	// Inputs Outputs
	Digital_Inputs_NrOfObjects			: ST_CAN_Object := (Name:='Digital Inputs_NrOfObjects',				Index:=16#21C0,					Length:=1, 	Default_Value:=14);
	Digital_Inputs_Digital_Input_1		: ST_CAN_Object := (Name:='Digital Inputs_Digital Input 1',			Index:=16#21C0,	Subindex:=1,	Length:=2);
	Digital_Inputs_Digital_Input_2		: ST_CAN_Object := (Name:='Digital Inputs_Digital Input 2',			Index:=16#21C0,	Subindex:=2,	Length:=2);
	Digital_Inputs_Digital_Input_3		: ST_CAN_Object := (Name:='Digital Inputs_Digital Input 3',			Index:=16#21C0,	Subindex:=3,	Length:=2);
	Digital_Inputs_Digital_Input_4		: ST_CAN_Object := (Name:='Digital Inputs_Digital Input 4',			Index:=16#21C0,	Subindex:=4,	Length:=2);
	Digital_Inputs_Digital_Input_5		: ST_CAN_Object := (Name:='Digital Inputs_Digital Input 5',			Index:=16#21C0,	Subindex:=5,	Length:=2);
	Digital_Inputs_Digital_Input_6		: ST_CAN_Object := (Name:='Digital Inputs_Digital Input 6',			Index:=16#21C0,	Subindex:=6,	Length:=2);
	Digital_Inputs_Digital_Input_7		: ST_CAN_Object := (Name:='Digital Inputs_Digital Input 7',			Index:=16#21C0,	Subindex:=7,	Length:=2);
	Digital_Inputs_Digital_Input_8		: ST_CAN_Object := (Name:='Digital Inputs_Digital Input 8',			Index:=16#21C0,	Subindex:=8,	Length:=2);
	Digital_Inputs_Watchdog_Input		: ST_CAN_Object := (Name:='Digital Inputs_Watchdog Input',			Index:=16#21C0,	Subindex:=9,	Length:=2);
	Digital_Inputs_Watchdog_Control		: ST_CAN_Object := (Name:='Digital Inputs_Watchdog Control',		Index:=16#21C0,	Subindex:=10,	Length:=2);
	Digital_Inputs_Watchdog_Fault		: ST_CAN_Object := (Name:='Digital Inputs_Watchdog Fault',			Index:=16#21C0,	Subindex:=11,	Length:=2);
	Digital_Inputs_PWM_enabled			: ST_CAN_Object := (Name:='Digital Inputs_PWM enabled',				Index:=16#21C0,	Subindex:=12,	Length:=2);
	Digital_Inputs_STO_L				: ST_CAN_Object := (Name:='Digital Inputs_STO_L',					Index:=16#21C0,	Subindex:=13,	Length:=2);
	Digital_Inputs_HW_ID				: ST_CAN_Object := (Name:='Digital Inputs_HW ID',					Index:=16#21C0,	Subindex:=14,	Length:=2);
	Digital_Outputs_NrOfObjects			: ST_CAN_Object := (Name:='Digital Outputs_NrOfObjects',			Index:=16#21C1,					Length:=1,						Default_Value:=3);
	Digital_Outputs_Digital_Output_1	: ST_CAN_Object := (Name:='Digital Outputs_Digital Output 1',		Index:=16#21C1,	Subindex:=1,	Length:=2);
	Digital_Outputs_Digital_Output_2	: ST_CAN_Object := (Name:='Digital Outputs_Digital Output 2',		Index:=16#21C1,	Subindex:=2,	Length:=2);
	Digital_Outputs_Digital_Output_3	: ST_CAN_Object := (Name:='Digital Outputs_Digital Output 3',		Index:=16#21C1,	Subindex:=3,	Length:=2);
	Analog_Inputs_NrOfObjects			: ST_CAN_Object := (Name:='Analog Inputs_NrOfObjects',				Index:=16#21C2,					Length:=1,						Default_Value:=2);
	Analog_Inputs_Analog_In_1			: ST_CAN_Object := (Name:='Analog Inputs_Analog In 1',				Index:=16#21C2,	Subindex:=1,	Length:=2);
	Analog_Inputs_Analog_In_2			: ST_CAN_Object := (Name:='Analog Inputs_Analog In 2',				Index:=16#21C2,	Subindex:=2,	Length:=2);
	
	// Temperature
	Drive_temperature					: ST_CAN_Object := (Name:='Drive temperature', 						Index:=16#2200,					Length:=2);
	Motor_temperature					: ST_CAN_Object := (Name:='Motor temperature', 						Index:=16#2202,					Length:=2);
	
	// HEM Reset
	BiSS_Encoder_Reset					: ST_CAN_Object := (Name:='BiSS Encoder Reset', 					Index:=16#3502,					Length:=1);
	
	// Time
	Time_since_power_on					: ST_CAN_Object := (Name:='Time since power on', 					Index:=16#4008);
	
	// CAN parameters
	CAN_open_Settings_NrOfObjects		: ST_CAN_Object := (Name:='CAN open Settings_NrOfObjects', 			Index:=16#400A,					Length:=1, 						Default_Value:=2);
	CAN_open_Settings_Node_Id			: ST_CAN_Object := (Name:='CAN open Settings_Node Id', 				Index:=16#400A,	Subindex:=1,	Length:=1,	RPDO_Mappable:=TRUE,Default_Value:=2);
	CAN_open_Settings_Baud_rate			: ST_CAN_Object := (Name:='CAN open Settings_Baud rate', 			Index:=16#400A,	Subindex:=2,	Length:=1,	RPDO_Mappable:=TRUE,Default_Value:=0);
	
	// Reset
	Reset								: ST_CAN_Object := (Name:='Reset', 									Index:=16#400B,					Length:=2);
	
	// Error, warning, message
	Error_Warning_status_NrOfObjects					: ST_CAN_Object := (Name:='Error Warning status_NrOfObjects', 						Index:=16#4080,					Length:=1, Default_Value:=2);
	Error_Warning_status_Error_count					: ST_CAN_Object := (Name:='Error Warning status_Error count', 						Index:=16#4080,	Subindex:=1);
	Error_Warning_status_Warning_count					: ST_CAN_Object := (Name:='Error Warning status_Warning count', 					Index:=16#4080,	Subindex:=2);
	Message_History_NrOfObjects							: ST_CAN_Object := (Name:='Message History_NrOfObjects', 							Index:=16#4081,					Length:=1, Default_Value:=6);
	Message_History_Rx_Last_address						: ST_CAN_Object := (Name:='Message History_Rx Last address', 						Index:=16#4081,	Subindex:=1);
	Message_History_Rx_Last_message_data				: ST_CAN_Object := (Name:='Message History_Rx Last message data', 					Index:=16#4081,	Subindex:=2);
	Message_History_Rx_2nd_Last_address					: ST_CAN_Object := (Name:='Message History_Rx 2nd Last address', 					Index:=16#4081,	Subindex:=3);
	Message_History_Rx_2nd_Last_message_data			: ST_CAN_Object := (Name:='Message History_Rx 2nd Last message data',				Index:=16#4081,	Subindex:=4);
	Message_History_Rx_3rd_Last_address					: ST_CAN_Object := (Name:='Message History_Rx 3rd Last address', 					Index:=16#4081,	Subindex:=5);
	Message_History_Rx_3rd_Last_message_data			: ST_CAN_Object := (Name:='Message History_Rx 3rd Last message data',				Index:=16#4081,	Subindex:=6);
	Error_history_device_time_NrOfObjects				: ST_CAN_Object := (Name:='Error history device time_NrOfObjects',					Index:=16#4082,					Length:=1, Default_Value:=4);
	Error_history_device_time_Field_1					: ST_CAN_Object := (Name:='Error history device time_Field 1', 						Index:=16#4082,	Subindex:=1);
	Error_history_device_time_Field_2					: ST_CAN_Object := (Name:='Error history device time_Field 2', 						Index:=16#4082,	Subindex:=2);
	Error_history_device_time_Field_3					: ST_CAN_Object := (Name:='Error history device time_Field 3', 						Index:=16#4082,	Subindex:=3);
	Error_history_device_time_Field_4					: ST_CAN_Object := (Name:='Error history device time_Field 4', 						Index:=16#4082,	Subindex:=4);
	Manufacturer_Error_Message_and_Code_NrOfObjects		: ST_CAN_Object := (Name:='Manufacturer Error Message and Code_NrOfObjects', 		Index:=16#4083,					Length:=1, Default_Value:=8);
	Manufacturer_Error_Message_and_Code_Field_1_Message	: ST_CAN_Object := (Name:='Manufacturer Error Message and Code_Field 1 Message', 	Index:=16#4083,	Subindex:=1);
	Manufacturer_Error_Message_and_Code_Field_1_Code	: ST_CAN_Object := (Name:='Manufacturer Error Message and Code_Field 1 Code', 		Index:=16#4083,	Subindex:=2,	Length:=2);
	Manufacturer_Error_Message_and_Code_Field_2_Message	: ST_CAN_Object := (Name:='Manufacturer Error Message and Code_Field 2 Message', 	Index:=16#4083,	Subindex:=3);
	Manufacturer_Error_Message_and_Code_Field_2_Code	: ST_CAN_Object := (Name:='Manufacturer Error Message and Code_Field 2 Code', 		Index:=16#4083,	Subindex:=4,	Length:=2);
	Manufacturer_Error_Message_and_Code_Field_3_Message	: ST_CAN_Object := (Name:='Manufacturer Error Message and Code_Field 3 Message', 	Index:=16#4083,	Subindex:=5);
	Manufacturer_Error_Message_and_Code_Field_3_Code	: ST_CAN_Object := (Name:='Manufacturer Error Message and Code_Field 3 Code', 		Index:=16#4083,	Subindex:=6,	Length:=2);
	Manufacturer_Error_Message_and_Code_Field_4_Message	: ST_CAN_Object := (Name:='Manufacturer Error Message and Code_Field 4 Message', 	Index:=16#4083,	Subindex:=7);
	Manufacturer_Error_Message_and_Code_Field_4_Code	: ST_CAN_Object := (Name:='Manufacturer Error Message and Code_Field 4 Code', 		Index:=16#4083,	Subindex:=8,	Length:=2);
	Warning_Code_NrOfObjects							: ST_CAN_Object := (Name:='Warning Code_NrOfObjects', 								Index:=16#408A, 				Length:=1, Default_Value:=4);
	Warning_Code_Field_1								: ST_CAN_Object := (Name:='Warning Code_Field 1', 									Index:=16#408A,	Subindex:=1, 	Length:=2);
	Warning_Code_Field_2								: ST_CAN_Object := (Name:='Warning Code_Field 2', 									Index:=16#408A,	Subindex:=2, 	Length:=2);
	Warning_Code_Field_3								: ST_CAN_Object := (Name:='Warning Code_Field 3', 									Index:=16#408A,	Subindex:=3, 	Length:=2);
	Warning_Code_Field_4								: ST_CAN_Object := (Name:='Warning Code_Field 4', 									Index:=16#408A,	Subindex:=4, 	Length:=2);
	Warning_history_device_time_NrOfObjects				: ST_CAN_Object := (Name:='Warning history device time_NrOfObjects', 				Index:=16#408B, 				Length:=1, Default_Value:=4);
	Warning_history_device_time_Field_1					: ST_CAN_Object := (Name:='Warning history device time_Field 1', 					Index:=16#408B,	Subindex:=1);
	Warning_history_device_time_Field_2					: ST_CAN_Object := (Name:='Warning history device time_Field 2', 					Index:=16#408B,	Subindex:=2);
	Warning_history_device_time_Field_3					: ST_CAN_Object := (Name:='Warning history device time_Field 3', 					Index:=16#408B,	Subindex:=3);
	Warning_history_device_time_Field_4					: ST_CAN_Object := (Name:='Warning history device time_Field 4', 					Index:=16#408B,	Subindex:=4);
	Errors_Warnings_Version								: ST_CAN_Object := (Name:='Errors/Warnings Version', 								Index:=16#40BF, 				Length:=2);
END_VAR

// ---- GVLs/PDO.TcGVL
{attribute 'qualified_only'}
VAR_GLOBAL
	// Values for RPDOs
	Controlword 				AT%Q*: WORD 				:= 0;
	Mode_of_operation 			AT%Q*: E_Mode_of_Operation 	:= E_Mode_of_Operation.No_mode_active;
	Target_velocity		 		AT%Q*: DINT 				:= 0;
	Profile_velocity			AT%Q*: DINT					:= 0;
	Target_position		 		AT%Q*: DINT					:= 0;
	Target_torque		 		AT%Q*: INT					:= 0;
	vl_target_velocity	 		AT%Q*: INT					:= 0;
	
		
	// Values from TPDOs
	Statusword 					AT%I*: WORD					:= 0;
	Mode_of_operation_display	AT%I*: E_Mode_of_Operation 	:= E_Mode_of_Operation.No_mode_active;
	DC_link_circuit_voltage		AT%I*: DWORD				:= 0;
	Current_actual_value		AT%I*: INT					:= 0;
	Velocity_actual_value 		AT%I*: DINT					:= 0;
	Position_actual_value 		AT%I*: DINT					:= 0;
	Torque_actual_value 		AT%I*: INT					:= 0;
	Drive_temperature			AT%I*: INT					:= 0;
	Motor_temperature			AT%I*: INT					:= 0;
	vl_Velocity_actual_value 		AT%I*: INT					:= 0;	
END_VAR

// ---- POUs/MAIN.TcPOU
PROGRAM MAIN
VAR		
	State			: INT			:= 255;
	
	Controlmode		: E_Controlmode;
	
	Current_State	: E_Statemachine_State;
	Target_State	: E_Statemachine_State;
		
	bTaster1 AT%I*	: BOOL;
	bTaster2 AT%I*	: BOOL;
	bTaster3 AT%I*	: BOOL;
	bTaster4 AT%I*	: BOOL;
	bTaster5 AT%I*	: BOOL;
	bTaster6 AT%I*	: BOOL;
	bTaster7 AT%I*	: BOOL;
	bTaster8 AT%I*	: BOOL;
	bTaster1_Flanke	: R_TRIG;
	bTaster2_Flanke	: R_TRIG;
	bTaster3_Flanke	: R_TRIG;
	bTaster4_Flanke	: R_TRIG;
	bTaster5_Flanke	: R_TRIG;
	bTaster6_Flanke	: R_TRIG;
	bTaster7_Flanke	: R_TRIG;
	bTaster8_Flanke	: R_TRIG;
	
	
	bLED1 	AT%Q* 	: BOOL;
	bLED2 	AT%Q* 	: BOOL;
	bLED3 	AT%Q* 	: BOOL;
	bLED4 	AT%Q* 	: BOOL;
	bLED5 	AT%Q* 	: BOOL;
	bLED6 	AT%Q* 	: BOOL;
	bLED7 	AT%Q* 	: BOOL;
	bLED8 	AT%Q* 	: BOOL;
	
	CAN_Object_Testing		: FB_DS402_Object_Testing;
			
	Profile_Position_Mode	: Profile_Position_Mode;
	
	READ_Manufacturer_label	: READ_Manufacturer_label;
	
	Encoder_Alignment		: Encoder_Alignment;
	
	Homing_parameters		: ST_Homing_parameters;
	Homing_mode				: Homing_Mode;
	
	NodeID			: BYTE := 2;
	
	Data		: ARRAY [0..255] OF BYTE;
	
	SDO_READ		: FB_SDO_READ;
	ReadStart		: BOOL;
	ReadError		: DWORD;
	ReadData		: ARRAY [0..255] OF BYTE;
	
	SDO_WRITE		: FB_SDO_WRITE;
	WriteData		: ARRAY [0..255] OF BYTE;
	WriteStart		: BOOL;
	WriteError		: DWORD;

	Start_Testing	: FB_Sequenz_Testing;
	
	Position_set	: BOOL;
	
	Position_1		: DINT 	:= 0;
	Position_2		: DINT	:= 16#10000;

	Start_Merker	: BOOL;
	Finished		: BOOL;
	i				: DINT;
	
	STOP			: BOOL;
	
	Quick_Stop		: BOOL := FALSE;
	
	New_Controlword	: WORD;
		
	Fehler: DWORD;
	
	Startsequence 	: ARRAY [0..12] OF E_Test_step 	:= [E_Test_step.Switch_on_disabled,															
														E_Test_step.Velocity_window_30rpm,
														E_Test_step.Velocity_window_100ms,	
														E_Test_step.Mode_PVM,
														E_Test_step.Acceleration_1000,
														E_Test_step.Deceleration_1000,
														E_Test_step.PVM_Velocity_1000,
														E_Test_step.Ready_to_switch_on,
														E_Test_step.Switched_on,
														E_Test_step.Operation_enabled,
														E_Test_step.Wait_1000ms, 
														E_Test_step.Check_Statusword_Target_reached_200ms, 
														E_Test_step.Switch_on_disabled];
	
	Stop_Testing_SM : J_Stop_Testing_SM;
	Temp_Control_Word : WORD;
END_VAR

// Determine state
Current_State := GET_STATE(PDO.Statusword);
(*
// Show State with LEDs on IO module
bLED1 := (Current_State = E_Statemachine_State.Not_ready_to_switch_on);
bLED2 := (Current_State = E_Statemachine_State.Switch_on_disabled);
bLED3 := (Current_State = E_Statemachine_State.Ready_to_switch_on);
bLED4 := (Current_State = E_Statemachine_State.Switched_on);
bLED5 := (Current_State = E_Statemachine_State.Operation_enabled);
bLED6 := (Current_State = E_Statemachine_State.Quick_stop_active);
bLED7 := (Current_State = E_Statemachine_State.Fault_reaction_active);
bLED8 := (Current_State = E_Statemachine_State.Fault);

// Stop condition is all taster off
STOP := NOT bTaster1 AND NOT bTaster2 AND NOT bTaster3 AND NOT bTaster4 AND NOT bTaster5 AND NOT bTaster6 AND NOT bTaster7 AND NOT bTaster8;

// Reset if all taster are high
IF bTaster1 AND bTaster2 AND bTaster3 AND bTaster4 AND bTaster5 AND bTaster6 AND bTaster7 AND bTaster8 THEN
	State := 0;
END_IF

// Detect rising egdes
bTaster1_Flanke(CLK := bTaster1);
bTaster2_Flanke(CLK := bTaster2);
bTaster3_Flanke(CLK := bTaster3);
bTaster4_Flanke(CLK := bTaster4);
bTaster5_Flanke(CLK := bTaster5);	
bTaster6_Flanke(CLK := bTaster6);
bTaster7_Flanke(CLK := bTaster7);
bTaster8_Flanke(CLK := bTaster8);

*)
New_Controlword := PDO.Controlword;
Temp_Control_Word := New_Controlword;

//Stop Testing Added by Jan

	IF NOT Stop_Testing_SM.Finished THEN
		Stop_Testing_SM( JST_NodeID := NodeID,
					     JST_Start_Testing := TRUE,
						 JST_Current_State := Current_State,
						 JST_Controlword => New_Controlword);
						   
	END_IF



// Logger
GLB.Logger();
(*	


CASE State OF	
	// ********** Initial steps **********	
	0: // Idle
		CASE Controlmode OF
			E_controlmode.IO_Testmode:
				// In this mode the function are startet by digital inputs.		
				Target_State 			:= E_statemachine_state.Switch_on_disabled;
				PDO.Mode_of_operation 	:= E_Mode_of_operation.No_mode_active;
			
				IF NOT Stop THEN
					IF 		bTaster1_Flanke.Q 	THEN	
						// ************** Object test **************	
						State := 10;							
					
					ELSIF 	bTaster2_Flanke.Q 	THEN	
						// ********* Test the Start Testing ********
						State := 40;


					//ELSIF 	bTaster2_Flanke.Q 	THEN							
						// ********** Velocity Mode **********	
						//PDO.Mode_of_operation 	:= E_Mode_of_operation.Velocity_mode;
						//Target_State 			:= E_statemachine_state.Operation_enabled;
						//PDO.vl_target_velocity 	:= 1000;
						//State := 1;
						
					ELSIF 	bTaster3_Flanke.Q 	THEN
						// ********** Profile Velocity Mode **********			
						PDO.Mode_of_operation 	:= E_Mode_of_operation.Profile_velocity_mode;
						Target_State 			:= E_statemachine_state.Operation_enabled;
						PDO.Target_velocity 	:= 100000;			
						State := 1;
			
					ELSIF 	bTaster4_Flanke.Q 	THEN
						// ********** Profile Position Mode **********	
						PDO.Mode_of_operation 	:= E_Mode_of_operation.Profile_position_mode;
						Target_State 			:= E_statemachine_state.Operation_enabled;
						PDO.Profile_velocity 	:= 1000000;						
						PDO.Target_position 	:= Position_1;	
						Start_Merker 			:= TRUE;
						State := 1;
						
					ELSIF 	bTaster5_Flanke.Q 	THEN
						// ********** Profile Position Mode **********	
						PDO.Mode_of_operation 	:= E_Mode_of_operation.Profile_position_mode;
						Target_State 			:= E_statemachine_state.Operation_enabled;
						PDO.Profile_velocity 	:= 100000;
						PDO.Target_position 	:= Position_2;	
						Start_Merker 			:= TRUE;
						State := 1;
						
					//ELSIF 	bTaster6_Flanke.Q 	THEN  
						// ************* Homing mode **************		
					//	Homing_parameters.Homing_mode := E_Homing_mode.Homing_on_current_position;			
					//	State := 20;				
						
					ELSIF 	bTaster6_Flanke.Q 	THEN	
						// Open / Close Logger File				
						IF GLB.Logger.IsOpen THEN 
							GLB.Logger(CloseFlag := TRUE);
						ELSE
							GLB.Logger(OpenFlag := TRUE);				
						END_IF								
					
					ELSIF 	bTaster7_Flanke.Q	THEN
						// Test: Write Logger Message						
						GLB.Logger(Message:= 'Hallo');	

					ELSIF 	bTaster8_Flanke.Q	THEN
						// Test: Save Logger Message						
						GLB.Logger(SaveFlag := TRUE);
						
					END_IF			
				END_IF					
				New_Controlword := CONTROLWORD_STATE_CHANGE(Current_State, Target_State);	
						
				
			E_Controlmode.Manual:
				// The user have to set the pdo values or the target state manually.
				State := 255;
			
		END_CASE
		
		
	1: // Start process
		IF 	STOP THEN	
			Target_State := E_statemachine_state.Switch_on_disabled;
			State := 3;	
		ELSIF Current_State = E_statemachine_state.Operation_enabled THEN 	
			State := 2;			
		END_IF;		
	
		New_Controlword := CONTROLWORD_STATE_CHANGE(Current_State, Target_State);	
				
		
	2: // Mode specific
		New_Controlword := CONTROLWORD_STATE_CHANGE(Current_State, Target_State);
	
		CASE PDO.Mode_of_operation OF				
			E_Mode_of_operation.Profile_position_mode:
				Profile_Position_Mode(Current_State:=Current_State, Statusword:=PDO.Statusword, Controlword:=New_Controlword, Start:=Start_Merker, Finished=>Finished);
				
				
		END_CASE
				
		IF STOP THEN 
			Target_State := E_statemachine_state.Switch_on_disabled;
			New_Controlword := CONTROLWORD_STATE_CHANGE(Current_State, Target_State);	
			State := 3; 
		END_IF
					
		
	3:	// Stop process
		Target_State := E_statemachine_state.Switch_on_disabled;	
		New_Controlword := CONTROLWORD_STATE_CHANGE(Current_State, Target_State);			
		IF Current_State = E_statemachine_state.Switch_on_disabled THEN	State := 0;	END_IF
		
		
	10:	// ********** CAN Object Testing **********	
		CAN_Object_Testing(Start := TRUE);	
		State := State + 1;

	11: // Wait for finish
		CAN_Object_Testing(Start := FALSE);		
		IF CAN_Object_Testing.Finished AND STOP THEN	
			State := 0;	
		END_IF
			
		
	20:	// ************* Homing mode **************
		Homing_mode(NodeID:=NodeID, Start:=TRUE, Current_State:=Current_State, Statusword:=PDO.Statusword, Homing_parameters:=Homing_parameters, Controlword=>New_Controlword, Mode_of_operation=>PDO.Mode_of_operation);
		State := State + 1;
	
	21: // Wait for finish
		Homing_mode(Start:=FALSE, Current_State:=Current_State, Statusword:=PDO.Statusword, Controlword=>New_Controlword);	
		IF Homing_mode.Finished THEN
			State := 0;
		END_IF
		
		
	30:	// ********** Encoder Alignment ***********	
		Encoder_Alignment(Start:=TRUE, Current_State:=Current_State, Statusword:=PDO.Statusword, Controlword=>New_Controlword);
		State := State + 1;
	
	31: // Wait for finish
		Encoder_Alignment(Start:=FALSE, Current_State:=Current_State, Statusword:=PDO.Statusword, Controlword=>New_Controlword);	
		IF Encoder_Alignment.Finished THEN
			State := 0;
		END_IF

		
	40:	// Test the Start Testing		
		Start_Testing(Start:=TRUE, Sequence_Name:='Test Sequence', Step_list:=Startsequence);
		State := State + 1;
	
	41: // Wait for finish
		Start_Testing(Start:=FALSE);
		New_Controlword := PDO.Controlword;		
		IF Start_Testing.Finished THEN
			State := 0;
		END_IF

		
	255: // **************** Init *****************
		GLB.Logger(OpenFlag:=TRUE);
		State := 0;
	
		
	ELSE	// Reset to Idle
		State := 0;
	
END_CASE	
*)

// Write the new Controlword
PDO.Controlword := New_Controlword;

END_PROGRAM

// ---- POUs/CAN_Object_Testing.TcPOU
FUNCTION_BLOCK CAN_Object_Testing
VAR_INPUT
	NodeID			: BYTE; (* This Port No. addresses the CANopen Node (see System Manager) *)
	Start			: BOOL;
END_VAR
VAR_OUTPUT
	Finished		: BOOL;
END_VAR
VAR_IN_OUT
	CAN_Objects		: ARRAY [*] OF ST_CAN_Object;
END_VAR
VAR
	State			: BYTE := 0;
	Index			: DINT := 0;
	i				: BYTE := 0;
	
	Data		: ARRAY [0..255] OF BYTE;
	
	NMT_WRITE		: FB_NMT_WRITE;
	SDO_READ		: FB_SDO_READ;
	SDO_WRITE		: FB_SDO_WRITE;	
			
	RPDO_Nr				: BYTE := 3;	
	RPDO_Current_Number	: BYTE := 0;
	RPDO_Current_Mapped	: DWORD := 0;	
	
	TPDO_Nr				: BYTE := 3;
	TPDO_Current_Number	: BYTE := 0;
	TPDO_Current_Mapped	: DWORD := 0;
END_VAR

IF Start AND State = 255 THEN 
	State := 0;
END_IF

SDO_READ(StartReading:=FALSE);
SDO_WRITE(StartWriting:=FALSE);
NMT_WRITE(StartWriting:=FALSE);


CASE State OF	
	// ********** Initial steps **********	
	0: // NMT Set to Preoperational
		IF Start THEN
			NMT_WRITE(
				AdsNetID	:= GLB.ADSNetID_CAN,
				PortNr		:= 16#1000 + GLB.NodeID,
				ADSSTATE	:= ADSSTATE_RUN, 
				DEVSTATE	:= 0,
				StartWriting:=TRUE			
			);	
			State := State + 1;			
		END_IF
		
	1: // Wait for finish			
			IF NMT_WRITE.WriteDataFinished THEN
				Index := 0;	
				State := State + 1;	
			END_IF

			
	2:	// RPDO disable
		Data[3] := 16#80;
		Data[2] := 0;			
		Data[1] := RPDO_Nr + 1;
		Data[0] := NodeID;	
			
		SDO_WRITE(
			ADSNetID		:= GLB.ADSNetID_CAN,
			PortNr 		 	:= 16#1000 + GLB.NodeID,
			CO_Index 	 	:= 16#1400 + RPDO_Nr,
			CO_SubIndex  	:= 1,
			DataLength 	 	:= 4,
			StartWriting 	:= TRUE,
			WriteData 	 	:= Data );
		State := State + 1;	
		
	3: // Wait for finish
		IF SDO_WRITE.WriteDataFinished THEN
			State := State + 1;
		END_IF	
		
		
	4:	// RPDO Current Number of mapped objects
		SDO_READ(
			ADSNetID		:= GLB.ADSNetID_CAN,				
			PortNr 		 	:= 16#1000 + GLB.NodeID,
			CO_Index 		:= 16#1600 + RPDO_Nr,
			CO_SubIndex 	:= 0,
			DataLength 		:= 1,
			StartReading	:= TRUE	);
		State := State + 1;	
		
	5: // Wait for finish
		IF SDO_READ.ReadDataAvailable THEN
			RPDO_Current_Number := SDO_READ.ReadData[0];
			State := State + 1;
		END_IF
		
	
	6:	// RPDO Current mapped object
		SDO_READ(
			ADSNetID		:= GLB.ADSNetID_CAN,				
			PortNr 		 	:= 16#1000 + GLB.NodeID,
			CO_Index 		:= 16#1600 + RPDO_Nr,
			CO_SubIndex 	:= 1,
			DataLength 		:= 4,
			StartReading	:= TRUE);
		State := State + 1;	
		
	7: // Wait for finish
		IF SDO_READ.ReadDataAvailable THEN
			RPDO_Current_Mapped := SHL(BYTE_TO_DWORD(SDO_READ.ReadData[3]),24) + SHL(BYTE_TO_DWORD(SDO_READ.ReadData[2]),16) + SHL(BYTE_TO_DWORD(SDO_READ.ReadData[1]),8) + BYTE_TO_DWORD(SDO_READ.ReadData[0]);								
			State := State + 1;
		END_IF		
			
		
	8:	// TPDO disable
		Data[3] := 16#80;
		Data[2] := 0;			
		Data[1] := TPDO_Nr;
		Data[0] := NodeID + 16#80;	
			
		SDO_WRITE(
			ADSNetID		:= GLB.ADSNetID_CAN,
			PortNr 		 	:= 16#1000 + GLB.NodeID,
			CO_Index 	 	:= 16#1800 + TPDO_Nr,
			CO_SubIndex  	:= 1,
			DataLength 	 	:= 4,
			StartWriting 	:= TRUE,
			WriteData 	 	:= Data );		
		State := State + 1;	
		
	9: // Wait for finish
		IF SDO_WRITE.WriteDataFinished THEN
			State := State + 1;
		END_IF	
		

	10:	// TPDO Current Number of mapped objects
		SDO_READ(
			ADSNetID		:= GLB.ADSNetID_CAN,				
			PortNr 		 	:= 16#1000 + GLB.NodeID,
			CO_Index 		:= 16#1A00 + TPDO_Nr,
			CO_SubIndex 	:= 0,
			DataLength 		:= 1,
			StartReading	:= TRUE	);		
		State := State + 1;	
		
	11: // Wait for finish
		IF SDO_READ.ReadDataAvailable THEN
			TPDO_Current_Number := SDO_READ.ReadData[0];			
			State := State + 1;
		END_IF
		

	12:	// TPDO Current mapped object
		SDO_READ(
			ADSNetID		:= GLB.ADSNetID_CAN,				
			PortNr 		 	:= 16#1000 + GLB.NodeID,
			CO_Index 		:= 16#1A00 + TPDO_Nr,
			CO_SubIndex 	:= 1,
			DataLength 		:= 4,
			StartReading	:= TRUE	);		
		State := State + 1;	
		
	13: // Wait for finish
		IF SDO_READ.ReadDataAvailable THEN
			TPDO_Current_Mapped := SHL(BYTE_TO_DWORD(SDO_READ.ReadData[3]),24) + SHL(BYTE_TO_DWORD(SDO_READ.ReadData[2]),16) + SHL(BYTE_TO_DWORD(SDO_READ.ReadData[1]),8) + BYTE_TO_DWORD(SDO_READ.ReadData[0]);							
			State := 16;
		END_IF		
		
		
		
	// ********** Test steps **********
	16:	// Init
		IF CAN_Objects[Index].Length_Tested THEN 
			CAN_Objects[Index].Length_Tested := FALSE;
			CAN_Objects[Index].Length_Error := 0;
		ELSE
			CAN_Objects[Index].Length_Target := CAN_Objects[Index].Length; 
		END_IF
		
		IF CAN_Objects[Index].Readable_Tested THEN 
			CAN_Objects[Index].Readable_Tested := FALSE;
			CAN_Objects[Index].Readable_Error := 0;
			CAN_Objects[Index].Read_Value := 0;
		ELSE
			CAN_Objects[Index].Readable_Target := CAN_Objects[Index].Readable;
		END_IF
		
		IF CAN_Objects[Index].Writable_Tested THEN 
	    	CAN_Objects[Index].Writable_Tested := FALSE;
			CAN_Objects[Index].Writable_Error := 0; 
			CAN_Objects[Index].Write_Value := 0;
		ELSE		
			CAN_Objects[Index].Writable_Target := CAN_Objects[Index].Writable;
		END_IF
				
		IF CAN_Objects[Index].RPDO_Mappable_Tested THEN 
	    	CAN_Objects[Index].RPDO_Mappable_Tested := FALSE;
			CAN_Objects[Index].RPDO_Mappable_Error := 0; 
		ELSE		
			CAN_Objects[Index].RPDO_Mappable_Target := CAN_Objects[Index].RPDO_Mappable;
		END_IF
		
		IF CAN_Objects[Index].TPDO_Mappable_Tested THEN 
	    	CAN_Objects[Index].TPDO_Mappable_Tested := FALSE;
			CAN_Objects[Index].TPDO_Mappable_Error := 0; 
		ELSE		
			CAN_Objects[Index].TPDO_Mappable_Target := CAN_Objects[Index].TPDO_Mappable;
		END_IF	

		State := State + 1;
			
		
	17:	// Read Test
		SDO_READ(
			ADSNetID		:= GLB.ADSNetID_CAN,				
			PortNr 		 	:= 16#1000 + GLB.NodeID,
			CO_Index 		:= CAN_Objects[Index].Index,
			CO_SubIndex 	:= CAN_Objects[Index].Subindex,
			DataLength 		:= CAN_Objects[Index].Length,
			StartReading	:= TRUE	);		
		State := State + 1;
		
	18: // Read Test, wait for finish
		IF SDO_READ.ReadDataAvailable THEN
			CAN_Objects[Index].Readable_Tested := TRUE;
			CAN_Objects[Index].Read_Value := SHL(BYTE_TO_DWORD(SDO_READ.ReadData[3]),24) + SHL(BYTE_TO_DWORD(SDO_READ.ReadData[2]),16) + SHL(BYTE_TO_DWORD(SDO_READ.ReadData[1]),8) + BYTE_TO_DWORD(SDO_READ.ReadData[0]);	
			CAN_Objects[Index].Readable_Error := SDO_READ.Error;
			
			// LENGTH setzen !!!	
								
			State := State + 1;
		END_IF
	
		
	19:	// Write Test
		IF CAN_Objects[Index].Write_Value_Usage THEN CAN_Objects[Index].Write_Value := CAN_Objects[Index].Read_Value; END_IF
		FOR i := 0 TO CAN_Objects[Index].Length - 1 DO
			Data[i] := DWORD_TO_BYTE(SHR(CAN_Objects[Index].Write_Value, (8*i)));
		END_FOR;
			
		SDO_WRITE(
			ADSNetID	:= GLB.ADSNetID_CAN,
			PortNr 		 := 16#1000 + GLB.NodeID,
			CO_Index 	 := CAN_Objects[Index].Index,
			CO_SubIndex  := CAN_Objects[Index].Subindex,
			DataLength 	 := CAN_Objects[Index].Length,
			StartWriting := TRUE,
			WriteData 	 := Data );		
		State := State + 1;
			
	20: // Write Test, wait for finish
		IF SDO_WRITE.WriteDataFinished THEN
			CAN_Objects[Index].Writable_Tested := TRUE;
			CAN_Objects[Index].Write_Value := SHL(BYTE_TO_DWORD(SDO_Write.WriteData[3]),24) + SHL(BYTE_TO_DWORD(SDO_Write.WriteData[2]),16) + SHL(BYTE_TO_DWORD(SDO_Write.WriteData[1]),8) + BYTE_TO_DWORD(SDO_Write.WriteData[0]);				
			CAN_Objects[Index].Writable_Error := SDO_WRITE.Error;
			
			
			// Falls Read-Test nicht erfolgreich -> LENGTH hier setzen !!!	
			
		
			State := State + 1;
		END_IF

		
	21: // RPDO test	
		Data[0] := CAN_Objects[Index].Length * 8;
		Data[1] := CAN_Objects[Index].SubIndex;
		Data[2] := DWORD_TO_BYTE(CAN_Objects[Index].Index);
		Data[3] := DWORD_TO_BYTE(SHR(CAN_Objects[Index].Index,8));
			
		SDO_WRITE(
			ADSNetID	:= GLB.ADSNetID_CAN,
			PortNr 		 := 16#1000 + GLB.NodeID,
			CO_Index 	 := 16#1600 + RPDO_Nr,
			CO_SubIndex  := 1,
			DataLength 	 := 4,
			StartWriting := TRUE,
			WriteData 	 := Data );	
		State := State + 1;
			
	22: // RPDO test, wait for finish
		IF SDO_WRITE.WriteDataFinished THEN
			CAN_Objects[Index].RPDO_Mappable_Tested := TRUE;
			CAN_Objects[Index].RPDO_Mappable_Error := SDO_WRITE.Error;
									
			State := State + 1;
		END_IF	

				
	23: // TPDO test
		// Value for TPDO test is the same like RPDO test
 
		SDO_WRITE(
			ADSNetID	:= GLB.ADSNetID_CAN,
			PortNr 		 := 16#1000 + GLB.NodeID,
			CO_Index 	 := 16#1A00 + TPDO_Nr,
			CO_SubIndex  := 1,
			DataLength 	 := 4,
			StartWriting := TRUE,
			WriteData 	 := Data );	
		State := State + 1;
			
	24: // TPDO test, wait for finish
		IF SDO_WRITE.WriteDataFinished THEN
			CAN_Objects[Index].TPDO_Mappable_Tested := TRUE;
			CAN_Objects[Index].TPDO_Mappable_Error := SDO_WRITE.Error;
			
			State := State + 1;
		END_IF
		
		
	25: // Next object
		CAN_Objects[Index].Error := (CAN_Objects[Index].Readable_Error > 0) OR (CAN_Objects[Index].Writable_Error > 0) OR (CAN_Objects[Index].RPDO_Mappable_Error > 0) OR (CAN_Objects[Index].TPDO_Mappable_Error > 0);
			
		IF Index < UPPER_BOUND(CAN_Objects,1) THEN
			Index := Index + 1;
			State := 16;
		ELSE
			State := 128;
		END_IF
	
		
	// ********** Ending steps **********		
	128: // RPDO Reset mapped object
		Data[0] := DWORD_TO_BYTE(RPDO_Current_Mapped);
		Data[1] := DWORD_TO_BYTE(SHR(RPDO_Current_Mapped,8));
		Data[2] := DWORD_TO_BYTE(SHR(RPDO_Current_Mapped,16));
		Data[3] := DWORD_TO_BYTE(SHR(RPDO_Current_Mapped,24));
		SDO_WRITE(
			ADSNetID		:= GLB.ADSNetID_CAN,			
			PortNr 		 	:= 16#1000 + GLB.NodeID,
			CO_Index 		:= 16#1600 + TPDO_Nr,
			CO_SubIndex 	:= 1,
			DataLength 		:= 4,
			StartWriting	:= TRUE,
			WriteData 	 	:= Data );
		State := State + 1;
			
	129: // RPDO Reset mapped object, wait for finish		
		IF SDO_WRITE.WriteDataFinished THEN
			State := State + 1;
		END_IF		
			
		
	130: // RPDO Reset Number of mapped objects
		Data[0] := RPDO_Current_Number;
			
		SDO_WRITE(
			ADSNetID		:= GLB.ADSNetID_CAN,
			PortNr 		 	:= 16#1000 + GLB.NodeID,
			CO_Index 		:= 16#1600 + RPDO_Nr,
			CO_SubIndex 	:= 0,
			DataLength 		:= 1,
			StartWriting 	:= TRUE,
			WriteData 	 	:= Data );
		State := State + 1;
			
	131: // RPDO Reset Number of mapped objects, wait for finish			
		IF SDO_WRITE.WriteDataFinished THEN
			State := State + 1;
		END_IF			

		
	132: // RPDO reactivate
		Data[3] := 0;
		Data[2] := 0;			
		Data[1] := RPDO_Nr + 1;
		Data[0] := NodeID;	
			
		SDO_WRITE(
			ADSNetID	:= GLB.ADSNetID_CAN,
			PortNr 		 := 16#1000 + GLB.NodeID,
			CO_Index 	 := 16#1400 + RPDO_Nr,
			CO_SubIndex  := 1,
			DataLength 	 := 4,
			StartWriting := TRUE,
			WriteData 	 := Data );
		State := State + 1;
			
	133: // RPDO reactivate, wait for finish	
		IF SDO_WRITE.WriteDataFinished THEN
			State := State + 1;
		END_IF	
		
		
	134: // TPDO Reset mapped object
		Data[0] := DWORD_TO_BYTE(TPDO_Current_Mapped);
		Data[1] := DWORD_TO_BYTE(SHR(TPDO_Current_Mapped,8));
		Data[2] := DWORD_TO_BYTE(SHR(TPDO_Current_Mapped,16));
		Data[3] := DWORD_TO_BYTE(SHR(TPDO_Current_Mapped,24));
		
		SDO_WRITE(
			ADSNetID		:= GLB.ADSNetID_CAN,			
			PortNr 		 	:= 16#1000 + GLB.NodeID,
			CO_Index 		:= 16#1A00 + TPDO_Nr,
			CO_SubIndex 	:= 1,
			DataLength 		:= 4,
			StartWriting	:= TRUE,
			WriteData 	 	:= Data );
		State := State + 1;
			
	135: // TPDO Reset mapped object, wait for finish	
		IF SDO_WRITE.WriteDataFinished THEN
			State := State + 1;
		END_IF			
			
		
	136:// TPDO Reset Number of mapped objects
		Data[0] := TPDO_Current_Number;
			
		SDO_WRITE(
			ADSNetID		:= GLB.ADSNetID_CAN,
			PortNr 		 	:= 16#1000 + GLB.NodeID,
			CO_Index 		:= 16#1A00 + RPDO_Nr,
			CO_SubIndex 	:= 0,
			DataLength 		:= 1,
			StartWriting 	:= TRUE,
			WriteData 	 	:= Data );
		State := State + 1;
			
	137: // TPDO Reset Number of mapped objects, wait for finish	
		IF SDO_WRITE.WriteDataFinished THEN
			State := State + 1;
		END_IF			

		
	138: // TPDO reactivate
		Data[3] := 0;
		Data[2] := 0;			
		Data[1] := TPDO_Nr;
		Data[0] := NodeID + 16#80;	
			
		SDO_WRITE(
			ADSNetID	:= GLB.ADSNetID_CAN,
			PortNr 		 := 16#1000 + GLB.NodeID,
			CO_Index 	 := 16#1400 + RPDO_Nr,
			CO_SubIndex  := 1,
			DataLength 	 := 4,
			StartWriting := TRUE,
			WriteData 	 := Data );
		State := State + 1;
			
	139: // TPDO reactivate, wait for finish	
		IF SDO_WRITE.WriteDataFinished THEN
			State := State + 1;
		END_IF	
						
	
	140: // NMT Set to operational
		NMT_WRITE(
			ADSNetID	:= GLB.ADSNetID_CAN,
			PORTNr		:= 16#1000 + GLB.NodeID,
			ADSSTATE	:= ADSSTATE_RUN,
			DEVSTATE	:= 1,
			StartWriting:=TRUE );	
		State := State + 1;
			
	141: // RPDO Reset Number of mapped objects, wait for finish	
		IF NMT_WRITE.WriteDataFinished THEN
			State := 255;	
		END_IF

		
	// ********** End **********
	ELSE	// Tests finished	
		Finished := TRUE;
		State := 255;
			
END_CASE

END_FUNCTION_BLOCK

// ---- POUs/FB/Basic/FB_NMT_WRITE.TcPOU
FUNCTION_BLOCK FB_NMT_WRITE
VAR_INPUT
	ADSNetID		: STRING(23); 	(* The AMSNetID addresses the EL6751. Can be empty if only one local single channel card is present*)
	PortNr			: WORD; 		(* The Port No. addresses the CANopen Node (see System Manager) *)
	ADSSTATE		: UINT; 		(* This is the value of the ADS state (ADSSTATE_RUN (=5) or ADSSTATE_STOP (=6)*)
	DEVSTATE		: UINT;			(* This is the value of the wanted device state (ADSSTATE_RUN -> 1 = OP, 0 = PREOP or ADSSTATE_STOP -> 0 = STOP)*)
	StartWriting	: BOOL; 		(* only reset to FALSE after WriteDataFinished=TRUE*)
END_VAR
VAR_OUTPUT
	WriteDataFinished	: BOOL;
	Error			: DWORD;
END_VAR
VAR
	state			: BYTE := 0;
	ADSWRTCTL		: ADSWRTCTL;
	NMTData			: ARRAY[0..1] OF BYTE; (*This array contains the data to be written to the CANopen Object	Dictionary*)
END_VAR

CASE
state OF
0:
	IF StartWriting THEN
		WriteDataFinished := FALSE;
		Error := 0;
		ADSWRTCTL(
			NetID		:= ADSNetID,
			PORT		:= PortNr,
			ADSSTATE	:= ADSSTATE,
			DEVSTATE	:= DEVSTATE,
			LEN			:= 2,
			SRCADDR		:= ADR(NMTData),
			WRITE		:= TRUE,
			TMOUT 		:= T#100MS
		);	
		IF ADSWRTCTL.err THEN
			state := 2;
			WriteDataFinished := TRUE;
			Error := ADSWRTCTL.ErrId;
		ELSE
			state := 1;
		END_IF
	ELSE
		ADSWRTCTL(
			NetID		:= ADSNetID,
			PORT		:= PortNr,
			ADSSTATE	:= ADSSTATE, 
			DEVSTATE	:= DEVSTATE,
			LEN			:= 2, 
			SRCADDR		:= ADR(NMTData),
			WRITE		:= FALSE,
			TMOUT 		:= T#1S
		);
	END_IF
	
1:
	ADSWRTCTL(WRITE:= FALSE);
	IF ADSWRTCTL.err THEN
		state := 2;
		WriteDataFinished := TRUE;
		Error := ADSWRTCTL.ErrId;
	ELSE
		IF NOT ADSWRTCTL.busy THEN
			state := 2;
			WriteDataFinished := TRUE;
		END_IF
	END_IF
	
2:
	ADSWRTCTL(WRITE:= FALSE);
	state := 0;
END_CASE

END_FUNCTION_BLOCK

// ---- POUs/FB/Basic/FB_SDO_READ.TcPOU
FUNCTION_BLOCK FB_SDO_READ
VAR_INPUT
	ADSNetID		: STRING(23); 	(* The AMSNetID addresses the EL6751. Can be empty if only one local single channel card is present*)
	PortNr			: WORD;	 		(* This Port No. addresses the CANopen Node (see System Manager) *)
	CO_Index		: DWORD; 		(* This is the Index of the CANopen Object Dictionary Entry*)
	CO_SubIndex		: DWORD; 		(* This is the Sub-Index of the CANopen Object Dictionary Entry*)
	DataLength		: DWORD; 		(* This is the Length of the CANopen Object Dictionary Entry*)
	StartReading	: BOOL;  		(* only reset to FALSE after ReadDataAvailable=TRUE*)
END_VAR
VAR_OUTPUT
	ReadData		: ARRAY[0..255] OF BYTE;
	ReadDataAvailable	: BOOL;
	Error			: DWORD;
END_VAR
VAR
	state			: BYTE 	:= 0;
	ADSREAD			: ADSREAD;
END_VAR

CASE
state OF
0:
	IF StartReading THEN
		ReadDataAvailable := FALSE;
		Error := 0;
		ADSRead(
			NETID		:= ADSNetID,
			PORT		:= PortNr,
			IDXGRP		:= CO_Index,
			IDXOFFS		:= CO_SubIndex,
			LEN			:= DataLength,
			DESTADDR	:= ADR(ReadData),
			READ		:= TRUE,
			TMOUT		:= T#100MS
		);

		IF ADSRead.err THEN
			state := 2;
			ReadDataAvailable := TRUE;
			Error := ADSRead.ErrId;
		ELSE
			state := 1;
		END_IF
	ELSE
		ADSRead(
			NETID		:= ADSNetID,
			PORT		:= PortNr,
			IDXGRP		:= CO_Index,
			IDXOFFS		:= CO_SubIndex,
			LEN			:= DataLength,
			DESTADDR	:= ADR(ReadData),
			READ		:= FALSE,
			TMOUT 		:= T#100MS
		);
	END_IF
	
1:
	ADSRead(READ:= FALSE);
	IF ADSRead.err THEN
		state := 2;
		ReadDataAvailable := TRUE;
		Error := ADSRead.ErrId;
	ELSE
		IF NOT ADSRead.busy THEN
			state := 2;
			ReadDataAvailable := TRUE;
		END_IF
	END_IF
	
2:
	ADSRead(READ:= FALSE);
	state := 0;
	
END_CASE

END_FUNCTION_BLOCK

// ---- POUs/FB/Basic/FB_SDO_WRITE.TcPOU
FUNCTION_BLOCK FB_SDO_WRITE
VAR_INPUT
	ADSNetID		: STRING(23); 	(* The AMSNetID addresses the EL6751. Can be empty if only one local single channel card is present*)
	PortNr			: WORD; 		(* The Port No. addresses the CANopen Node (see System Manager) *)
	CO_Index		: DWORD; 		(* This is the Index of the CANopen Object Dictionary Entry*)
	CO_SubIndex		: DWORD; 		(* This is the Sub-Index of the CANopen Object Dictionary Entry*)
	DataLength		: DWORD; 		(* This is the Length of the CANopen Object Dictionary Entry*)
	StartWriting	: BOOL; 		(* only reset to FALSE after WriteDataFinished=TRUE*)
	WriteData		: ARRAY[0..255] OF BYTE; (*This array contains the data to be written to the CANopen Object	Dictionary*)
END_VAR
VAR_OUTPUT
	WriteDataFinished	: BOOL;
	Error			: DWORD;
END_VAR
VAR
	state			: BYTE := 0;
	ADSWRITE		: ADSWRITE;
END_VAR

CASE
state OF
0:
	IF StartWriting THEN
		WriteDataFinished := FALSE;
		Error := 0;
		ADSWrite(
			NETID	:= ADSNetID,
			PORT	:= PortNr,
			IDXGRP	:= CO_Index,
			IDXOFFS	:= CO_SubIndex,
			LEN		:= DataLength,
			SRCADDR	:= ADR(WriteData),
			WRITE	:= TRUE,
			TMOUT 	:= T#100MS
		);
		IF ADSWrite.err THEN
			state := 2;
			WriteDataFinished := TRUE;
			Error := ADSWrite.ErrId;
		ELSE
			state := 1;
		END_IF
	ELSE
		ADSWrite(
			NETID	:= '',
			PORT	:= PortNr,
			IDXGRP	:= CO_Index,
			IDXOFFS	:= CO_SubIndex,
			LEN		:= DataLength,
			SRCADDR	:= ADR(WriteData),
			WRITE	:= FALSE,
			TMOUT 	:= T#100MS
		);
	END_IF
	
1:
	ADSWrite(WRITE:= FALSE);
	IF ADSWrite.err THEN
		state := 2;
		WriteDataFinished := TRUE;
		Error := ADSWrite.ErrId;
	ELSE
		IF NOT ADSWrite.busy THEN
			state := 2;
			WriteDataFinished := TRUE;
		END_IF
	END_IF
	
2:
	ADSWrite(WRITE:= FALSE);
	state := 0;
END_CASE

END_FUNCTION_BLOCK

// ---- POUs/FB/FB_DS402_Object_Testing.TcPOU
FUNCTION_BLOCK FB_DS402_Object_Testing
VAR_INPUT
	Start			: BOOL;
END_VAR
VAR_OUTPUT
	Finished		: BOOL;
	Error			: BOOL := FALSE;
END_VAR
VAR
	State			: BYTE := 0;
	Index			: DINT := 0;
	
	NMT_WRITE		: FB_NMT_WRITE;
	
	SDO_READ		: FB_SDO_READ;
	ReadData		: ARRAY [0..255] OF BYTE;
	
	SDO_WRITE		: FB_SDO_WRITE;
	WriteData		: ARRAY [0..255] OF BYTE;		
			
	RPDO_Nr				: BYTE := 3;	
	RPDO_Current_Number	: BYTE := 0;
	RPDO_Current_Mapped	: DWORD := 0;	
	
	TPDO_Nr				: BYTE := 3;
	TPDO_Current_Number	: BYTE := 0;
	TPDO_Current_Mapped	: DWORD := 0;
	
	
	Object_List_Testing	: FB_Object_List_Testing;
	
	
	Objects_general			: ARRAY [0..11] OF ST_CAN_Object := [DS402_Object_List.Abort_connection_option_code,
																 DS402_Object_List.Error_code,
																 DS402_Object_List.Controlword,
																 DS402_Object_List.Statusword,
																 DS402_Object_List.Quick_stop_option_code,
																 DS402_Object_List.Shutdown_option_code,
																 DS402_Object_List.Disable_operation_option_code,
																 DS402_Object_List.Halt_option_code,
																 DS402_Object_List.Fault_reaction_option_code,
																 DS402_Object_List.Modes_of_operation,
																 DS402_Object_List.Modes_of_operation_display,
																 DS402_Object_List.Supported_drive_modes];
		
	Objects_Factor_group	: ARRAY [0..25] OF ST_CAN_Object := [DS402_Object_List.Position_encoder_resolution_Highest_sub_index_supported,
																 DS402_Object_List.Position_encoder_resolution_Encoder_increments,
																 DS402_Object_List.Position_encoder_resolution_Motor_revolutions,
																 DS402_Object_List.Velocity_encoder_resolution_Highest_sub_index_supported,
																 DS402_Object_List.Velocity_encoder_resolution_Encoder_increments,
																 DS402_Object_List.Velocity_encoder_resolution_Motor_revolutions,
																 DS402_Object_List.Gear_ratio_Highest_sub_index_supported,
																 DS402_Object_List.Gear_ratio_Motor_shaft_revolutions,
																 DS402_Object_List.Gear_ratio_Driving_shaft_revolutions,
																 DS402_Object_List.Feed_constant_Highest_sub_index_supported,
																 DS402_Object_List.Feed_constant_Feed,
																 DS402_Object_List.Feed_constant_Shaft_Revolution,
																 DS402_Object_List.Velocity_Factor_Highest_sub_index_supported,
																 DS402_Object_List.Velocity_Factor_Numerator,
																 DS402_Object_List.Velocity_Factor_Divisor,
																 DS402_Object_List.Acceleration_Factor_Highest_sub_index_supported,
																 DS402_Object_List.Acceleration_Factor_Numerator,
																 DS402_Object_List.Acceleration_Factor_Divisor,
																 DS402_Object_List.Jerk_factor_Factor_Highest_sub_index_supported,
																 DS402_Object_List.Jerk_factor_Factor_Numerator,
																 DS402_Object_List.Jerk_factor_Factor_Divisor,
																 DS402_Object_List.Polarity,
																 DS402_Object_List.SI_unit_postion,
																 DS402_Object_List.SI_unit_velocity,
																 DS402_Object_List.SI_unit_acceleration,
																 DS402_Object_List.SI_unit_jerk];
							
	Objects_Position_control: ARRAY [0..10] OF ST_CAN_Object := [DS402_Object_List.Position_demand_value,
															 	 DS402_Object_List.Position_actual_internal_value,
																 DS402_Object_List.Position_actual_value,
																 DS402_Object_List.Following_error_window,
																 DS402_Object_List.Following_error_time_out,
																 DS402_Object_List.Position_window,
																 DS402_Object_List.Position_window_time,
																 DS402_Object_List.Position_option_code,
																 DS402_Object_List.Following_error_actual_value,
																 DS402_Object_List.Control_effort,
																 DS402_Object_List.Position_demand_integral_value];								
	
	Objects_PPM				: ARRAY [0..20] OF ST_CAN_Object := [DS402_Object_List.Target_position,
															 	 DS402_Object_List.Position_range_limit_Highest_sub_index_supported,
																 DS402_Object_List.Position_range_limit_Min_position_range_limit,
																 DS402_Object_List.Position_range_limit_Max_position_range_limit,
																 DS402_Object_List.Software_position_limit_Highest_sub_index_supported,
																 DS402_Object_List.Software_position_limit_Min_position_limit,
																 DS402_Object_List.Software_position_limit_Max_position_limit,
																 DS402_Object_List.Polarity,
																 DS402_Object_List.Max_profile_velocity,
																 DS402_Object_List.Profile_velocity,
																 DS402_Object_List.End_velocity,
																 DS402_Object_List.Profile_acceleration,
																 DS402_Object_List.Profile_deceleration,
																 DS402_Object_List.Quick_stop_deceleration,
																 DS402_Object_List.Motion_profile_type,
																 DS402_Object_List.Profile_jerk_use,
																 DS402_Object_List.Profile_jerk_Highest_sub_index_supported,
																 DS402_Object_List.Profile_jerk_1,
																 DS402_Object_List.Max_acceleration,
																 DS402_Object_List.Max_deceleration];

	Objects_VM				: ARRAY [0..20] OF ST_CAN_Object := [DS402_Object_List.vl_target_velocity,
															 	 DS402_Object_List.vl_velocity_demand,
															 	 DS402_Object_List.vl_velocity_actual_value,
															 	 DS402_Object_List.vl_velocity_min_max_amount_Highest_sub_index_supported,
															 	 DS402_Object_List.vl_velocity_min_max_amount_vl_velocity_min_amount,
															 	 DS402_Object_List.vl_velocity_min_max_amount_vl_velocity_max_amount,
															 	 DS402_Object_List.vl_velocity_acceleration_Highest_sub_index_supported,
															 	 DS402_Object_List.vl_velocity_acceleration_Delta_speed,
															 	 DS402_Object_List.vl_velocity_acceleration_Delta_time,
															 	 DS402_Object_List.vl_velocity_deceleration_Highest_sub_index_supported,
															 	 DS402_Object_List.vl_velocity_deceleration_Delta_speed,
															 	 DS402_Object_List.vl_velocity_deceleration_Delta_time,
															 	 DS402_Object_List.vl_velocity_quick_stop_Highest_sub_index_supported,
															 	 DS402_Object_List.vl_velocity_quick_stop_Delta_speed,
															 	 DS402_Object_List.vl_velocity_quick_stop_Delta_time,
															 	 DS402_Object_List.vl_set_point_factor_Highest_sub_index_supported,
															 	 DS402_Object_List.vl_set_point_factor_Numerator,
															 	 DS402_Object_List.vl_set_point_factor_Denominator,
															 	 DS402_Object_List.vl_dimension_factor_Highest_sub_index_supported,
															 	 DS402_Object_List.vl_dimension_factor_Numerator,
															 	 DS402_Object_List.vl_dimension_factor_Denominator];

	Objects_PVM				: ARRAY [0..16] OF ST_CAN_Object := [DS402_Object_List.Velocity_demand_value,
															 	 DS402_Object_List.Velocity_actual_value,
																 DS402_Object_List.Velocity_window,
																 DS402_Object_List.Velocity_window_time,
																 DS402_Object_List.Velocity_threshold,
																 DS402_Object_List.Velocity_threshold_time,
																 DS402_Object_List.Max_profile_velocity,
																 DS402_Object_List.Max_motor_speed,
																 DS402_Object_List.Profile_acceleration,
																 DS402_Object_List.Profile_deceleration,
																 DS402_Object_List.Quick_stop_deceleration,
																 DS402_Object_List.Motion_profile_type,
																 DS402_Object_List.Profile_jerk_Highest_sub_index_supported,
																 DS402_Object_List.Profile_jerk_1,
																 DS402_Object_List.Max_acceleration,
																 DS402_Object_List.Max_deceleration,
																 DS402_Object_List.Target_velocity];
	
	Objects_TM				: ARRAY [0..12] OF ST_CAN_Object := [DS402_Object_List.Target_torque,
															 	 DS402_Object_List.Max_torque,
															 	 DS402_Object_List.Max_current,
															 	 DS402_Object_List.Torque_demand,
															 	 DS402_Object_List.Motor_rated_current,
															 	 DS402_Object_List.Motor_rated_torque,
															 	 DS402_Object_List.Torque_actual_value,
															 	 DS402_Object_List.Current_actual_value,
															 	 DS402_Object_List.DC_link_circuit_voltage,
															 	 DS402_Object_List.Torque_slope,
															 	 DS402_Object_List.Torque_profile_type,
															 	 DS402_Object_List.Positive_torque_limit_value,
															 	 DS402_Object_List.Negative_torque_limit_value];
	
	Objects_HM				: ARRAY [0..7] OF ST_CAN_Object :=  [DS402_Object_List.Home_offset,
															 	 DS402_Object_List.Homing_method,
															 	 DS402_Object_List.Homing_speeds_Highest_sub_index_supported,
															 	 DS402_Object_List.Homing_speeds_Speed_during_search_for_switch,
															 	 DS402_Object_List.Homing_speeds_Speed_during_search_for_zero,
															 	 DS402_Object_List.Homing_acceleration,
															 	 DS402_Object_List.Supported_Homing_Methods_Highest_sub_index_supported,
															 	 DS402_Object_List.Supported_Homing_Methods_Supported_homing_method_1];

END_VAR

IF Start AND State = 255 THEN 
	Finished 	:= FALSE;	
	Error 		:= FALSE;
	State 		:= 0;
END_IF


SDO_READ(StartReading:=FALSE);
SDO_WRITE(StartWriting:=FALSE);
NMT_WRITE(StartWriting:=FALSE);
Object_List_Testing(Start:=FALSE);

CASE State OF	
	// ********** Initial steps **********	
	0: // NMT Set to Preoperational
		NMT_WRITE(
			AdsNetID	:= GLB.ADSNetID_CAN,
			PortNr		:= 16#1000 + GLB.NodeID,
			ADSSTATE	:= ADSSTATE_RUN, 
			DEVSTATE	:= 0,
			StartWriting:=TRUE			
		);	
		State := State + 1;	
					
	1: // Wait for finished
		IF NMT_WRITE.WriteDataFinished THEN
			Index := 0;	
			State := State + 1;	
		END_IF
		

	2:	// RPDO disable
		WriteData[3] := 16#80;
		WriteData[2] := 0;			
		WriteData[1] := RPDO_Nr + 1;
		WriteData[0] := GLB.NodeID;	
			
		SDO_WRITE(
			ADSNetID		:= GLB.ADSNetID_CAN,
			PortNr 		 	:= 16#1000 + GLB.NodeID,
			CO_Index 	 	:= 16#1400 + RPDO_Nr,
			CO_SubIndex  	:= 1,
			DataLength 	 	:= 4,
			StartWriting 	:= TRUE,
			WriteData 	 	:= WriteData );	
		State := State + 1;	
					
	3: // Wait for finished
		IF NMT_WRITE.WriteDataFinished THEN
			Index := 0;	
			State := State + 1;	
		END_IF
		
		
	4:	// RPDO Current Number of mapped objects
		SDO_READ(
			ADSNetID		:= GLB.ADSNetID_CAN,				
			PortNr 		 	:= 16#1000 + GLB.NodeID,
			CO_Index 		:= 16#1600 + RPDO_Nr,
			CO_SubIndex 	:= 0,
			DataLength 		:= 1,
			StartReading	:= TRUE	);	
		State := State + 1;	
					
	5: // Wait for finished
		IF SDO_READ.ReadDataAvailable THEN
			RPDO_Current_Number := SDO_READ.ReadData[0];
			State := State + 1;
		END_IF
		
		
	6:	// RPDO Number of mapped objects set to 0
		WriteData[3] := 0;
		WriteData[2] := 0;			
		WriteData[1] := 0;
		WriteData[0] := 0;	
		
		SDO_WRITE(
			ADSNetID		:= GLB.ADSNetID_CAN,
			PortNr 		 	:= 16#1000 + GLB.NodeID,
			CO_Index 	 	:= 16#1600 + RPDO_Nr,
			CO_SubIndex  	:= 0,
			DataLength 	 	:= 1,
			StartWriting 	:= TRUE,
			WriteData 	 	:= WriteData );	
		State := State + 1;	
					
	7: // Wait for finished
		IF NMT_WRITE.WriteDataFinished THEN
			Index := 0;	
			State := State + 1;	
		END_IF
				
		
	8:	// RPDO Current mapped object
		SDO_READ(
			ADSNetID		:= GLB.ADSNetID_CAN,				
			PortNr 		 	:= 16#1000 + GLB.NodeID,
			CO_Index 		:= 16#1600 + RPDO_Nr,
			CO_SubIndex 	:= 1,
			DataLength 		:= 4,
			StartReading	:= TRUE	);	
		State := State + 1;	
					
	9: // Wait for finished
		IF SDO_READ.ReadDataAvailable THEN
			RPDO_Current_Mapped := SHL(BYTE_TO_DWORD(SDO_READ.ReadData[3]),24) + SHL(BYTE_TO_DWORD(SDO_READ.ReadData[2]),16) + SHL(BYTE_TO_DWORD(SDO_READ.ReadData[1]),8) + BYTE_TO_DWORD(SDO_READ.ReadData[0]);								
			State := State + 1;
		END_IF		
			
		
	10:	// TPDO disable
		WriteData[3] := 16#80;
		WriteData[2] := 0;			
		WriteData[1] := TPDO_Nr;
		WriteData[0] := GLB.NodeID + 16#80;	
			
		SDO_WRITE(
			ADSNetID		:= GLB.ADSNetID_CAN,
			PortNr 		 	:= 16#1000 + GLB.NodeID,
			CO_Index 	 	:= 16#1800 + TPDO_Nr,
			CO_SubIndex  	:= 1,
			DataLength 	 	:= 4,
			StartWriting 	:= TRUE,
			WriteData 	 	:= WriteData );
		State := State + 1;	
					
	11: // Wait for finished
		IF SDO_WRITE.WriteDataFinished THEN
			State := State + 1;
		END_IF	
		

	12:	// TPDO Current Number of mapped objects
		SDO_READ(
			ADSNetID		:= GLB.ADSNetID_CAN,				
			PortNr 		 	:= 16#1000 + GLB.NodeID,
			CO_Index 		:= 16#1A00 + TPDO_Nr,
			CO_SubIndex 	:= 0,
			DataLength 		:= 1,
			StartReading	:= TRUE	);
		State := State + 1;	
					
	13: // Wait for finished
		IF SDO_READ.ReadDataAvailable THEN
			TPDO_Current_Number := SDO_READ.ReadData[0];			
			State := State + 1;
		END_IF
		
		
	14:	// RPDO Number of mapped objects set to 0
		WriteData[3] := 0;
		WriteData[2] := 0;			
		WriteData[1] := 0;
		WriteData[0] := 0;	
		
		SDO_WRITE(
			ADSNetID		:= GLB.ADSNetID_CAN,
			PortNr 		 	:= 16#1000 + GLB.NodeID,
			CO_Index 	 	:= 16#1A00 + RPDO_Nr,
			CO_SubIndex  	:= 0,
			DataLength 	 	:= 1,
			StartWriting 	:= TRUE,
			WriteData 	 	:= WriteData );	
		State := State + 1;	
					
	15: // Wait for finished
		IF NMT_WRITE.WriteDataFinished THEN
			Index := 0;	
			State := State + 1;	
		END_IF
					

	16:	// TPDO Current mapped object
		SDO_READ(
			ADSNetID		:= GLB.ADSNetID_CAN,				
			PortNr 		 	:= 16#1000 + GLB.NodeID,
			CO_Index 		:= 16#1A00 + TPDO_Nr,
			CO_SubIndex 	:= 1,
			DataLength 		:= 4,
			StartReading	:= TRUE	);
		State := State + 1;	
					
	17: // Wait for finished
		IF SDO_READ.ReadDataAvailable THEN
			TPDO_Current_Mapped := SHL(BYTE_TO_DWORD(SDO_READ.ReadData[3]),24) + SHL(BYTE_TO_DWORD(SDO_READ.ReadData[2]),16) + SHL(BYTE_TO_DWORD(SDO_READ.ReadData[1]),8) + BYTE_TO_DWORD(SDO_READ.ReadData[0]);							
			State := 32;
		END_IF		
		
		
		
	// ********** Test steps **********
	32:	// General objects
		Object_List_Testing(Object_List:=Objects_general, Start:=TRUE, Complete_test:=TRUE, RPDO_Nr:=RPDO_Nr, TPDO_Nr:=TPDO_Nr);
		State := State + 1;	
					
	33: // Wait for finished
		IF Object_List_Testing.Finished THEN
			Error := Error OR Object_List_Testing.error;
			State := State + 1;
		END_IF	
		
		
	34:	// Factor group objects
		Object_List_Testing(Object_List:=Objects_Factor_group, Start:=TRUE, Complete_test:=TRUE, RPDO_Nr:=RPDO_Nr, TPDO_Nr:=TPDO_Nr);
		State := State + 1;	
					
	35: // Wait for finished
		IF Object_List_Testing.Finished THEN
			Error := Error OR Object_List_Testing.error;
			State := State + 1;
		END_IF			
		
		
	36:	// Position control objects
		IF ((Objects_general[11].Read_Value AND 16#00C1) > 0) THEN
			Object_List_Testing(Object_List:=Objects_Position_control, Start:=TRUE, Complete_test:=TRUE, RPDO_Nr:=RPDO_Nr, TPDO_Nr:=TPDO_Nr);
			State := State + 1;	
		ELSE
			State := State + 2;
		END_IF	
					
	37: // Wait for finished
		IF Object_List_Testing.Finished THEN
			Error := Error OR Object_List_Testing.error;
			State := State + 1;
		END_IF	
	
		
	38:	// Profile Position Mode objects
		IF ((Objects_general[11].Read_Value AND 16#0001) > 16#0001) THEN	
			Object_List_Testing(Object_List:=Objects_PPM, Start:=TRUE, Complete_test:=TRUE, RPDO_Nr:=RPDO_Nr, TPDO_Nr:=TPDO_Nr);
			State := State + 1;	
		ELSE
			State := State + 2;
		END_IF	
			
	39: // Wait for finished
		IF Object_List_Testing.Finished THEN
			Error := Error OR Object_List_Testing.error;
			State := State + 1;
		END_IF	
	
		
	40:	// Velocity Mode objects
		IF ((Objects_general[11].Read_Value AND 16#0002) = 16#0002) THEN 	
			Object_List_Testing(Object_List:=Objects_VM, Start:=TRUE, Complete_test:=TRUE, RPDO_Nr:=RPDO_Nr, TPDO_Nr:=TPDO_Nr);
			State := State + 1;	
		ELSE
			State := State + 2;
		END_IF	
			
	41: // Wait for finished
		IF Object_List_Testing.Finished THEN
			Error := Error OR Object_List_Testing.error;
			State := State + 1;
		END_IF	
	
		
	42:	// Profile Velocity Mode objects
		IF ((Objects_general[11].Read_Value AND 16#0004) = 16#0004) THEN	
			Object_List_Testing(Object_List:=Objects_PVM, Start:=TRUE, Complete_test:=TRUE, RPDO_Nr:=RPDO_Nr, TPDO_Nr:=TPDO_Nr);
			State := State + 1;		
		ELSE
			State := State + 2;
		END_IF	
					
	43: // Wait for finished
		IF Object_List_Testing.Finished THEN
			Error := Error OR Object_List_Testing.error;
			State := State + 1;
		END_IF	
			
		
	44:	// Torque objects
		IF ((Objects_general[11].Read_Value AND 16#0008) = 16#0008) THEN 	
			Object_List_Testing(Object_List:=Objects_TM, Start:=TRUE, Complete_test:=TRUE, RPDO_Nr:=RPDO_Nr, TPDO_Nr:=TPDO_Nr);
			State := State + 1;		
		ELSE
			State := State + 2;
		END_IF	
					
	45: // Wait for finished
		IF Object_List_Testing.Finished THEN
			Error := Error OR Object_List_Testing.error;
			State := State + 1;
		END_IF	
		
		
	46:	// Homing Mode objects
		IF ((Objects_general[11].Read_Value AND 16#0020) = 16#0020) THEN
			Object_List_Testing(Object_List:=Objects_HM, Start:=TRUE, Complete_test:=TRUE, RPDO_Nr:=RPDO_Nr, TPDO_Nr:=TPDO_Nr);
			State := State + 1;		
		ELSE
			State := 96;
		END_IF	
					
	47: // Wait for finished
		IF Object_List_Testing.Finished THEN
			Error := Error OR Object_List_Testing.error;
			State := 96;
		END_IF	
			
				
		
	// ******** Restore values ********	
	96:	// RPDO Reset mapped object
		WriteData[0] := DWORD_TO_BYTE(RPDO_Current_Mapped);
		WriteData[1] := DWORD_TO_BYTE(SHR(RPDO_Current_Mapped,8));
		WriteData[2] := DWORD_TO_BYTE(SHR(RPDO_Current_Mapped,16));
		WriteData[3] := DWORD_TO_BYTE(SHR(RPDO_Current_Mapped,24));
		
		SDO_WRITE(
			ADSNetID		:= GLB.ADSNetID_CAN,			
			PortNr 		 	:= 16#1000 + GLB.NodeID,
			CO_Index 		:= 16#1600 + TPDO_Nr,
			CO_SubIndex 	:= 1,
			DataLength 		:= 4,
			StartWriting	:= TRUE,
			WriteData 	 	:= WriteData );
		State := State + 1;	
					
	97: // Wait for finished
		IF SDO_WRITE.WriteDataFinished THEN		
			State := State + 1;
		END_IF		
			
		
	98:	// RPDO Reset Number of mapped objects
		WriteData[0] := RPDO_Current_Number;
			
		SDO_WRITE(
			ADSNetID		:= GLB.ADSNetID_CAN,
			PortNr 		 	:= 16#1000 + GLB.NodeID,
			CO_Index 		:= 16#1600 + RPDO_Nr,
			CO_SubIndex 	:= 0,
			DataLength 		:= 1,
			StartWriting 	:= TRUE,
			WriteData 	 	:= WriteData );
		State := State + 1;	
					
	99: // Wait for finished
		IF SDO_WRITE.WriteDataFinished THEN
			State := State + 1;
		END_IF			

		
	100:	// RPDO reactivate
		WriteData[3] := 0;
		WriteData[2] := 0;			
		WriteData[1] := RPDO_Nr + 1;
		WriteData[0] := GLB.NodeID;	
	
		SDO_WRITE(
			ADSNetID	:= GLB.ADSNetID_CAN,
			PortNr 		 := 16#1000 + GLB.NodeID,
			CO_Index 	 := 16#1400 + RPDO_Nr,
			CO_SubIndex  := 1,
			DataLength 	 := 4,
			StartWriting := TRUE,
			WriteData 	 := WriteData );
		State := State + 1;	
					
	101: // Wait for finished
		IF SDO_WRITE.WriteDataFinished THEN
			State := State + 1;
		END_IF	
		
		
	102:	// TPDO Reset mapped object
		WriteData[0] := DWORD_TO_BYTE(TPDO_Current_Mapped);
		WriteData[1] := DWORD_TO_BYTE(SHR(TPDO_Current_Mapped,8));
		WriteData[2] := DWORD_TO_BYTE(SHR(TPDO_Current_Mapped,16));
		WriteData[3] := DWORD_TO_BYTE(SHR(TPDO_Current_Mapped,24));
		
		SDO_WRITE(
			ADSNetID		:= GLB.ADSNetID_CAN,			
			PortNr 		 	:= 16#1000 + GLB.NodeID,
			CO_Index 		:= 16#1A00 + TPDO_Nr,
			CO_SubIndex 	:= 1,
			DataLength 		:= 4,
			StartWriting	:= TRUE,
			WriteData 	 	:= WriteData );
		State := State + 1;	
					
	103: // Wait for finished
		IF SDO_WRITE.WriteDataFinished THEN
			State := State + 1;
		END_IF			
			
		
	104:	// TPDO Reset Number of mapped objects
		WriteData[0] := TPDO_Current_Number;
			
		SDO_WRITE(
			ADSNetID		:= GLB.ADSNetID_CAN,
			PortNr 		 	:= 16#1000 + GLB.NodeID,
			CO_Index 		:= 16#1A00 + RPDO_Nr,
			CO_SubIndex 	:= 0,
			DataLength 		:= 1,
			StartWriting 	:= TRUE,
			WriteData 	 	:= WriteData );
		State := State + 1;	
					
	105: // Wait for finished
		IF SDO_WRITE.WriteDataFinished THEN
			State := State + 1;
		END_IF			

		
	106:	// TPDO reactivate
		WriteData[3] := 0;
		WriteData[2] := 0;			
		WriteData[1] := TPDO_Nr;
		WriteData[0] := GLB.NodeID + 16#80;	
			
		SDO_WRITE(
			ADSNetID	:= GLB.ADSNetID_CAN,
			PortNr 		 := 16#1000 + GLB.NodeID,
			CO_Index 	 := 16#1400 + RPDO_Nr,
			CO_SubIndex  := 1,
			DataLength 	 := 4,
			StartWriting := TRUE,
			WriteData 	 := WriteData );
		State := State + 1;	
					
	107: // Wait for finished
		IF SDO_WRITE.WriteDataFinished THEN
			State := State + 1;
		END_IF	
						
	
	108: // NMT Set to operational
		NMT_WRITE(
			ADSNetID	:= GLB.ADSNetID_CAN,
			PORTNr		:= 16#1000 + GLB.NodeID,
			ADSSTATE	:= ADSSTATE_RUN,
			DEVSTATE	:= 1,
			StartWriting:=TRUE );	
		State := State + 1;	
					
	109: // Wait for finished
		IF NMT_WRITE.WriteDataFinished THEN
			State := 255;	
		END_IF
	
		
	// ************ Finished ************		
	255: // Tests finished
		Finished := TRUE;	
	

	ELSE		
		State := 255;
			
END_CASE

END_FUNCTION_BLOCK

// ---- POUs/FB/FB_Object_List_Testing.TcPOU
FUNCTION_BLOCK FB_Object_List_Testing
VAR_INPUT
	Start			: BOOL;	
	Complete_test	: BOOL := FALSE;	
	RPDO_Nr			: BYTE := 0;
	TPDO_Nr			: BYTE := 0;
END_VAR
VAR_IN_OUT
	Object_List		: ARRAY [*] OF ST_CAN_Object;
END_VAR
VAR_OUTPUT
	Finished		: BOOL := FALSE;
	Error			: BOOL := FALSE;
END_VAR
VAR
	State			: INT := 0;	
	Index 			: BYTE := 0;
	i 				: DINT := 0;
	
	Object_Testing	: FB_Object_Testing;

	SubIndex_Count	: BYTE := 0;
END_VAR

IF Start AND State = 255 THEN 
	Finished 	:= FALSE;
	Error 		:= FALSE;
	State 		:= 0;
END_IF


CASE State OF	
	0:	// Start check objects	
	IF Start THEN
		Object_Testing(CAN_Object:=Object_List[0], Start:=TRUE, Complete_test:=TRUE, RPDO_Nr:=3, TPDO_Nr:=3);
		Index := 0;
		
		State := State + 1;
	END_IF
	
	
	1:	// Running, wait for finish and start next object
	Object_Testing(CAN_Object:=Object_List[Index], Start:=FALSE);
	
	IF Object_Testing.Finished THEN
		
		CASE Object_List[Index].SubElements OF
			E_SubElement_types.With_fix_subelements:	// Object with fix subelements
				IF (Object_List[Index].Readable) AND ((Object_List[Index].Read_Value > 0) OR (Object_List[Index +1].Mandatory > 0)) THEN
					Index := Index + 1;
				ELSE
					Index := Index + 1 + DWORD_TO_BYTE(Object_List[Index].Default_Value);
				END_IF	 						
				
								
			E_SubElement_types.Fix_subelement:	// Next object
				Index := Index + 1;		
					
	
			E_SubElement_types.With_list:		// Object with a variable count of subelements	
				IF Object_List[Index].Readable AND Object_List[Index].Read_Value > 0 THEN
					Index := Index + 1;						
					Object_List[Index].Subindex := 1;
				ELSE
					Index := Index + 2;
				END_IF


			E_SubElement_types.List_element:	// Next variable subobject or next object
				IF Object_List[Index - 1].Read_Value > Object_List[Index].Subindex  THEN
					Object_List[Index].Subindex := Object_List[Index].Subindex + 1;
				ELSE
					Index := Index + 1;	
				END_IF
			
			
			E_SubElement_types.No:	// Standalone object -> next object
				Index := Index + 1;
					
	
			ELSE					// Unknown Type -> next object
				Index := Index + 1;
						
		END_CASE
		
		// Test next Object
		IF Index <= UPPER_BOUND(Object_List,1) THEN 
			Object_Testing(CAN_Object:=Object_List[Index], Start:=TRUE, Complete_test:=TRUE, RPDO_Nr:=3, TPDO_Nr:=3);	
		ELSE			
			State := 254;
		END_IF		
	END_IF	
	
	
	// ************ Finished ************			
	254: // Check error 
		Error := FALSE;
		FOR i := 0 TO UPPER_BOUND(Object_List,1) DO
			Error := Error OR Object_List[i].Error;			
		END_FOR;
		Finished := TRUE;	
		State := 255;
		
	255: // Tests finished
		Finished := TRUE;
	

	ELSE		
		State := 254;
		
END_CASE

END_FUNCTION_BLOCK

// ---- POUs/FB/FB_Object_Testing.TcPOU
FUNCTION_BLOCK FB_Object_Testing
VAR_INPUT
	Start			: BOOL;
	Complete_test	: BOOL := FALSE;	
	RPDO_Nr			: BYTE := 0;
	TPDO_Nr			: BYTE := 0;
END_VAR
VAR_IN_OUT
	CAN_Object		: ST_CAN_Object;	
END_VAR
VAR_OUTPUT
	Finished		: BOOL := FALSE;	
END_VAR
VAR
	State			: INT := 0;
	i				: BYTE;
	
	Data			: ARRAY [0..255] OF BYTE;	
	SDO_READ		: FB_SDO_READ;
	SDO_WRITE		: FB_SDO_WRITE;
	
	Message			: STRING(128);
END_VAR

IF Start AND State = 255 THEN 
	Finished 	:= FALSE;
	State 		:= 0;
END_IF


SDO_READ(StartReading:=FALSE);
SDO_WRITE(StartWriting:=FALSE);


CASE State OF	
	// ************** Init **************	
	0:	// Init
		IF Start THEN
			IF CAN_Object.Length_Tested THEN 
				CAN_Object.Length_Tested := FALSE;
				CAN_Object.Length_Error := 0;
			ELSE
				CAN_Object.Length_Target := CAN_Object.Length; 
			END_IF
			
			IF CAN_Object.Readable_Tested THEN 
				CAN_Object.Readable_Tested := FALSE;
				CAN_Object.Readable_Error := 0;
				CAN_Object.Read_Value := 0;
			ELSE
				CAN_Object.Readable_Target := CAN_Object.Readable;
			END_IF
			
			IF CAN_Object.Writable_Tested THEN 
				CAN_Object.Writable_Tested := FALSE;
				CAN_Object.Writable_Error := 0; 
			ELSE		
				CAN_Object.Writable_Target := CAN_Object.Writable;
			END_IF
					
			IF CAN_Object.RPDO_Mappable_Tested THEN 
				CAN_Object.RPDO_Mappable_Tested := FALSE;
				CAN_Object.RPDO_Mappable_Error := 0; 
			ELSE		
				CAN_Object.RPDO_Mappable_Target := CAN_Object.RPDO_Mappable;
			END_IF
			
			IF CAN_Object.TPDO_Mappable_Tested THEN 
				CAN_Object.TPDO_Mappable_Tested := FALSE;
				CAN_Object.TPDO_Mappable_Error := 0; 
			ELSE		
				CAN_Object.TPDO_Mappable_Target := CAN_Object.TPDO_Mappable;
			END_IF			
			
			Message := 'Check "';
			Message := CONCAT(Message, CAN_Object.Name);
			Message := CONCAT(Message, '" (0x');
			Message := CONCAT(Message, WORD_TO_HEXSTR(CAN_Object.Index, 4, FALSE));
			Message := CONCAT(Message, ', ');
			Message := CONCAT(Message, BYTE_TO_STRING(CAN_Object.SubIndex));
			Message := CONCAT(Message, ', ');
			Message := CONCAT(Message, BYTE_TO_STRING(CAN_Object.Length * 8));
			Message := CONCAT(Message, ' bits)');
				
			GLB.Logger(Message:=Message);
			
			State := State + 1;
		END_IF
		
		
	// ******* Read and write test ******	
	1:	// Read Test
		IF CAN_Object.Readable_Target OR Complete_Test THEN			
			SDO_READ(
				ADSNetID		:= GLB.ADSNetID_CAN,				
				PortNr 		 	:= 16#1000 + GLB.NodeID,
				CO_Index 		:= CAN_Object.Index,
				CO_SubIndex 	:= CAN_Object.Subindex,
				DataLength 		:= CAN_Object.Length_Target,
				ReadData		=> Data,
				StartReading	:= TRUE	);		
			State := State + 1;
		ELSE				
			State := State + 10;
		END_IF
			
	2: // Read test, wait for finish
		IF SDO_READ.ReadDataAvailable THEN
			CAN_Object.Readable_Tested := TRUE;
			CAN_Object.Readable_Error := SDO_READ.Error;
			CAN_Object.Readable := (CAN_Object.Readable_Error = 0);
			
			Message := 'Reading: ';
			IF CAN_Object.Readable = CAN_Object.Readable_Target THEN
				Message := CONCAT(Message, 'OK');
				IF CAN_Object.Readable THEN
					Message := CONCAT(Message, ' / readable');
				ELSE
					Message := CONCAT(Message, ' / not readable');						
				END_IF
			ELSE
				Message := CONCAT(Message, 'Error');	
				IF CAN_Object.Readable THEN
					Message := CONCAT(Message, ' / should not be readable');
				ELSE
					Message := CONCAT(Message, ' / should be readable');						
				END_IF	
			END_IF	
			GLB.Logger(Message:=Message);
			
			IF CAN_Object.Readable THEN			
				CAN_Object.Read_Value := SHL(BYTE_TO_DWORD(SDO_READ.ReadData[3]),24) + SHL(BYTE_TO_DWORD(SDO_READ.ReadData[2]),16) + SHL(BYTE_TO_DWORD(SDO_READ.ReadData[1]),8) + BYTE_TO_DWORD(SDO_READ.ReadData[0]);
	
				// If Reading is successful, the length is also correct.
				CAN_Object.Length_Tested := TRUE;	
				CAN_Object.Length := CAN_Object.Length_Target;
				CAN_Object.Length_Error := 0;								
			END_IF
								
			State := State + 9;
		END_IF
	
		
	11:	// Write Test
		IF CAN_Object.Writable_Target OR Complete_Test THEN
			// Use the read value for write value?
			IF CAN_Object.Write_Value_Usage THEN CAN_Object.Write_Value := CAN_Object.Read_Value; END_IF
			
			FOR i := 0 TO CAN_Object.Length - 1 DO
				Data[i] := DWORD_TO_BYTE(SHR(CAN_Object.Write_Value, (8*i)));			
			END_FOR;
			
			SDO_WRITE(
				ADSNetID	:= GLB.ADSNetID_CAN,
				PortNr 		 := 16#1000 + GLB.NodeID,
				CO_Index 	 := CAN_Object.Index,
				CO_SubIndex  := CAN_Object.Subindex,
				DataLength 	 := CAN_Object.Length_Target,
				WriteData 	 := Data,
				StartWriting := TRUE );		
			State := State + 1;
		ELSE
			State := State + 10;
		END_IF
		
	12: // Write test, wait for finish
		IF SDO_WRITE.WriteDataFinished THEN
			CAN_Object.Writable_Tested := TRUE;
			CAN_Object.Writable_Error := SDO_WRITE.Error;
			CAN_Object.Writable := (CAN_Object.Writable_Error = 0);

			Message := 'Writing: ';
			IF CAN_Object.Writable = CAN_Object.Writable_Target THEN
				Message := CONCAT(Message, 'OK');
				IF CAN_Object.Writable THEN
					Message := CONCAT(Message, ' / writable');
				ELSE
					Message := CONCAT(Message, ' / not writable');						
				END_IF
			ELSE
				Message := CONCAT(Message, 'Error');	
				IF CAN_Object.Writable THEN
					Message := CONCAT(Message, ' / should be not writable');
				ELSE
					Message := CONCAT(Message, ' / should be writable');						
				END_IF
			END_IF	
			GLB.Logger(Message:=Message);					
	
			IF CAN_Object.Writable THEN
				CAN_Object.Write_Value := SHL(BYTE_TO_DWORD(SDO_Write.WriteData[3]),24) + SHL(BYTE_TO_DWORD(SDO_Write.WriteData[2]),16) + SHL(BYTE_TO_DWORD(SDO_Write.WriteData[1]),8) + BYTE_TO_DWORD(SDO_Write.WriteData[0]);				
				
				// If Writing is successful, the length is also correct.
				CAN_Object.Length_Tested := TRUE;
				CAN_Object.Length := CAN_Object.Length_Target;			
				CAN_Object.Length_Error := 0;						
			END_IF
		
			State := State + 9;				
		END_IF
		
		
	21: // Analyse the readable and writable tests
			// The PDO tests make only sense, if the object exists. This means that it must be readable and/or writable.
			IF CAN_Object.Readable OR CAN_Object.Writable THEN
				// Go to PDO tests
				State := 101;
			ELSE	
				IF Complete_test THEN
					// Additional tests
					i := 1;
					State := State + 1;
				ELSE
					// Test is finished with error.
					State := 254;					
				END_IF					
			END_IF
		
	
	22: // Redo the read test with other length
		SDO_READ(
			ADSNetID		:= GLB.ADSNetID_CAN,				
			PortNr 		 	:= 16#1000 + GLB.NodeID,
			CO_Index 		:= CAN_Object.Index,
			CO_SubIndex 	:= CAN_Object.Subindex,
			DataLength 		:= i,
			ReadData		=> Data,
			StartReading	:= TRUE	);		
		State := State + 1;	
		
	23: // Read test, wait for finish
		IF SDO_READ.ReadDataAvailable THEN
			CAN_Object.Readable_Tested := TRUE;
			CAN_Object.Readable_Error := SDO_READ.Error;
			CAN_Object.Readable := (CAN_Object.Readable_Error = 0);
						
			IF CAN_Object.Readable THEN
				CAN_Object.Read_Value := SHL(BYTE_TO_DWORD(SDO_READ.ReadData[3]),24) + SHL(BYTE_TO_DWORD(SDO_READ.ReadData[2]),16) + SHL(BYTE_TO_DWORD(SDO_READ.ReadData[1]),8) + BYTE_TO_DWORD(SDO_READ.ReadData[0]);	

				// If Reading is successful, the correct length is found.
				CAN_Object.Length_Tested := TRUE;	
				CAN_Object.Length := i;
				IF i > CAN_Object.Length_Target THEN			
					CAN_Object.Length_Error := 16#06070012;	
					CAN_Object.Readable_Error := 16#06070012;					
				ELSIF i < CAN_Object.Length_Target THEN
					CAN_Object.Length_Error := 16#06070013;	
					CAN_Object.Readable_Error := 16#06070013;				
				END_IF
				
				State := State + 1;
				
			ELSE					
				// This length is also wrong, check next length or resume with write test
				CASE i OF	
					1:
						IF (CAN_Object.Length_Target = 2) THEN
							// next length is 4 byte							
							i := 4;
							State := State - 1;							
						ELSE
							// next length is 2 byte							
							i := 2;
							State := State - 1;	
						END_IF
						
					2:
						IF (CAN_Object.Length_Target = 4) THEN
							// Continue with write test
							i := 1;
							State := State + 1;
						ELSE
							// next length is 4 byte
							i := 4;
							State := State - 1;	
						END_IF						
	
					4:
						// Continue with write test
						i := 1;
						State := State + 1;
						
					ELSE
						// If i value is strange, continue with write test
						i := 1;						
						State := State + 1;		
				END_CASE					
			END_IF		
		END_IF

		
	24: // Redo the write test with other length
		SDO_WRITE(
			ADSNetID	:= GLB.ADSNetID_CAN,
			PortNr 		 := 16#1000 + GLB.NodeID,
			CO_Index 	 := CAN_Object.Index,
			CO_SubIndex  := CAN_Object.Subindex,
			DataLength 	 := i,
			WriteData 	 := Data,
			StartWriting := TRUE );		
		State := State + 1;	
		
	25: // Write test, wait for finish
		IF SDO_WRITE.WriteDataFinished THEN
			CAN_Object.Writable_Tested := TRUE;
			CAN_Object.Writable_Error := SDO_WRITE.Error;
			CAN_Object.Writable := (CAN_Object.Writable_Error = 0);
						
			IF CAN_Object.Writable THEN
				CAN_Object.Write_Value := SHL(BYTE_TO_DWORD(SDO_Write.WriteData[3]),24) + SHL(BYTE_TO_DWORD(SDO_Write.WriteData[2]),16) + SHL(BYTE_TO_DWORD(SDO_Write.WriteData[1]),8) + BYTE_TO_DWORD(SDO_Write.WriteData[0]);				
				
				// If Writing is successful, the length is also correct.
				CAN_Object.Length_Tested := TRUE;
				CAN_Object.Length := i;		

				IF i > CAN_Object.Length_Target THEN			
					IF (CAN_Object.Length_Error = 16#06070013) THEN CAN_Object.Length_Error := 16#06070010; ELSE CAN_Object.Length_Error := 16#06070012; END_IF	
					CAN_Object.Writable_Error := 16#06070012;					
				ELSIF i < CAN_Object.Length_Target THEN
					IF (CAN_Object.Length_Error = 16#06070012) THEN CAN_Object.Length_Error := 16#06070010; ELSE CAN_Object.Length_Error := 16#06070013; END_IF
					CAN_Object.Writable_Error := 16#06070013;				
				END_IF
				
				State := State + 1;
			ELSE					
				// This length is also wrong, check next length or resume with next step
				CASE i OF	
					1:
						IF (CAN_Object.Length_Target = 2) THEN
							// next length is 4 byte							
							i := 4;
							State := State - 1;	
						ELSE
							// next length is 2 byte							
							i := 2;
							State := State - 1;	
						END_IF
						
					2:
						IF (CAN_Object.Length_Target = 4) THEN
							// Continue with write test
							State := State + 1;
						ELSE
							// next length is 4 byte
							i := 4;
							State := State - 1;	
						END_IF						
	
					4:
						// Continue with write test
						State := State + 1;
						
					ELSE
						// If i value is strange, continue with write test
						i := 1;						
						State := State + 1;		
				END_CASE				
			END_IF		
		END_IF
	
		
	26: // If the object is now found, resume with the PDO tests. Otherwise the test is finished with error.
		IF CAN_Object.Readable OR CAN_Object.Writable THEN
			State := 101;	
		ELSE
			State := 254;
		END_IF	
		
		
	// *********** PDO Tests ************
	101: // RPDO test
		IF CAN_Object.RPDO_Mappable_Target OR Complete_Test THEN	
			Data[0] := CAN_Object.Length * 8;
			Data[1] := CAN_Object.SubIndex;
			Data[2] := DWORD_TO_BYTE(CAN_Object.Index);
			Data[3] := DWORD_TO_BYTE(SHR(CAN_Object.Index,8));
				
			SDO_WRITE(
				ADSNetID	:= GLB.ADSNetID_CAN,
				PortNr 		 := 16#1000 + GLB.NodeID,
				CO_Index 	 := 16#1600 + RPDO_Nr,
				CO_SubIndex  := 1,
				DataLength 	 := 4,
				StartWriting := TRUE,
				WriteData 	 := Data );	
			State := State + 1;
		ELSE			
			State := State + 10;
		END_IF
			
	102: // RPDO test, wait for finish
		IF SDO_WRITE.WriteDataFinished THEN
			CAN_Object.RPDO_Mappable_Tested := TRUE;
			CAN_Object.RPDO_Mappable_Error := SDO_WRITE.Error;
			CAN_Object.RPDO_Mappable := (CAN_Object.RPDO_Mappable_Error = 0);	
			
			Message := 'Mappable RPDO: ';
			IF CAN_Object.RPDO_Mappable = CAN_Object.RPDO_Mappable_Target THEN
				Message := CONCAT(Message, 'OK');
				IF CAN_Object.RPDO_Mappable THEN
					Message := CONCAT(Message, ' / mappable');
				ELSE
					Message := CONCAT(Message, ' / not mappable');						
				END_IF
			ELSE
				Message := CONCAT(Message, 'Error');	
				IF CAN_Object.RPDO_Mappable THEN
					Message := CONCAT(Message, ' / should be not mappable');
				ELSE
					Message := CONCAT(Message, ' / should be mappable');						
				END_IF
			END_IF	
			GLB.Logger(Message:=Message);								
		
			State := State + 9;
		END_IF	

				
	111: // TPDO test
		IF CAN_Object.RPDO_Mappable_Target OR Complete_Test THEN		
			Data[0] := CAN_Object.Length * 8;
			Data[1] := CAN_Object.SubIndex;
			Data[2] := DWORD_TO_BYTE(CAN_Object.Index);
			Data[3] := DWORD_TO_BYTE(SHR(CAN_Object.Index,8));
	 
			SDO_WRITE(
				ADSNetID	:= GLB.ADSNetID_CAN,
				PortNr 		 := 16#1000 + GLB.NodeID,
				CO_Index 	 := 16#1A00 + TPDO_Nr,
				CO_SubIndex  := 1,
				DataLength 	 := 4,
				StartWriting := TRUE,
				WriteData 	 := Data );				
			State := State + 1;
		ELSE
			State := 254;
		END_IF
			
	112: // TPDO test, wait for finish
		IF SDO_WRITE.WriteDataFinished THEN
			CAN_Object.TPDO_Mappable_Tested := TRUE;
			CAN_Object.TPDO_Mappable_Error := SDO_WRITE.Error;
			CAN_Object.TPDO_Mappable := (CAN_Object.TPDO_Mappable_Error = 0);	
				
			Message := 'Mappable TPDO: ';
			IF CAN_Object.TPDO_Mappable = CAN_Object.TPDO_Mappable_Target THEN
				Message := CONCAT(Message, 'OK');
				IF CAN_Object.TPDO_Mappable THEN
					Message := CONCAT(Message, ' / mappable');
				ELSE
					Message := CONCAT(Message, ' / not mappable');						
				END_IF
			ELSE
				Message := CONCAT(Message, 'Error');	
				IF CAN_Object.TPDO_Mappable THEN
					Message := CONCAT(Message, ' / should be not mappable');
				ELSE
					Message := CONCAT(Message, ' / should be mappable');						
				END_IF
			END_IF	
			GLB.Logger(Message:=Message);	
			
			State := 254;
		END_IF

		
	// ************ Finished ************	
	254: // Check error 
	IF (CAN_Object.Mandatory > 0) OR CAN_Object.Readable OR CAN_Object.Writable THEN
		CAN_Object.Error := ((CAN_Object.Readable <> CAN_Object.Readable_Target) OR (CAN_Object.Writable <> CAN_Object.Writable_Target) OR  
							(CAN_Object.RPDO_Mappable <> CAN_Object.RPDO_Mappable_Target) OR (CAN_Object.TPDO_Mappable <> CAN_Object.TPDO_Mappable_Target) OR
							(CAN_Object.Length <> CAN_Object.Length_Target));

		Message := 'Result: ';
		IF CAN_Object.Error THEN
			Message := CONCAT(Message, 'Error');
		ELSE				
			Message := CONCAT(Message, 'OK');
		END_IF	
		Message := CONCAT(Message, '$0A**********');		
		GLB.Logger(Message:=Message, SaveFlag:=TRUE);	
	ELSE
		// Optional object not exists
		Message := 'Result: OK / Optional object does not exist';	
		Message := CONCAT(Message, '$0A**********');		
		GLB.Logger(Message:=Message, SaveFlag:=TRUE);	
	
	END_IF
	
		Finished := TRUE;	
		State := 255;
		
	255: // Tests finished
		Finished := TRUE;	
	
	
	ELSE	
		State := 254;
		
END_CASE

END_FUNCTION_BLOCK

// ---- POUs/Profile_Position_Mode.TcPOU
FUNCTION_BLOCK Profile_Position_Mode
VAR_INPUT
	Current_State 	: E_Statemachine_State;	
	Statusword		: WORD;
END_VAR
VAR_IN_OUT
	Controlword 	: WORD;
	Start 			: BOOL;
END_VAR
VAR_OUTPUT
	Finished		: BOOL;
END_VAR
VAR
	Index 			: BYTE := 0;
END_VAR

IF Start THEN Index := 0; END_IF;

CASE Index OF	
	0: // Set Position
		IF (Statusword AND E_Statusword_Bits.PPM_Set_point_acknowledge) = E_Statusword_Bits.PPM_Set_point_acknowledge THEN
			Controlword := Controlword AND NOT E_Controlword_Bits.PPM_New_set_point;
			Index := 1;
		ELSE
			Controlword := Controlword OR E_Controlword_Bits.PPM_New_set_point;				
		END_IF
		
		
	1: // Position reached?
		FINISHED :=  ((Statusword AND E_Statusword_Bits.Target_reached) = E_Statusword_Bits.Target_reached);
						
END_CASE

END_FUNCTION_BLOCK

// ---- POUs/READ_Manufacturer_label.TcPOU
FUNCTION_BLOCK READ_Manufacturer_label
VAR_INPUT
	NodeID		: BYTE; (* This Port No. addresses the CANopen Node (see System Manager) *)	
	Start		: BOOL;
END_VAR
VAR_OUTPUT
	Label_Out	: ST_Manufacturer_label;
	Finished	: BOOL := FALSE;
END_VAR
VAR
	Index		: INT;
	Label		: ST_Manufacturer_label;
	SDO_READ 	: FB_SDO_READ;	
	SDO_READ_REAL 	: FB_SDO_READ_REAL;	
	SDO_WRITE 	: FB_SDO_WRITE;
	WriteData	: ARRAY [0..255] OF BYTE;		
	CAN_Objects	: INT;
END_VAR

// Restart after complete run
IF (Index = 255) AND Start THEN
	Index := 0;
END_IF


IF NOT (Index = 255) THEN 
	SDO_READ(StartReading:=FALSE);
	SDO_READ_REAL(StartReading:=FALSE);
END_IF
	
	
CASE Index OF	
	0: // Start reading Serial_Number
		IF Start THEN		
			Finished := FALSE;
			SDO_READ(	
				AdsNetID		:= GLB.ADSNetID_CAN,
				PortNr			:= 16#1000 + GLB.NodeID,
				CO_Index		:= 16#41C0,
				CO_SubIndex		:= 16#01,
				DataLength		:= 4,
				StartReading	:= TRUE	
			);	
			Index := Index + 1;
		END_IF
		
	1: // Serial_Number is read
		IF SDO_READ.ReadDataAvailable THEN
			Label.Serial_Number := SHL(BYTE_TO_DWORD(SDO_READ.ReadData[3]),24) + SHL(BYTE_TO_DWORD(SDO_READ.ReadData[2]),16) + SHL(BYTE_TO_DWORD(SDO_READ.ReadData[1]),8) + BYTE_TO_DWORD(SDO_READ.ReadData[0]);				
			Index := Index + 1;
		END_IF

	
	2: // Start reading Min_v
		SDO_READ(	
			AdsNetID		:= GLB.ADSNetID_CAN,
			PortNr			:= 16#1000 + GLB.NodeID,
			CO_Index		:= 16#41C0,
			CO_SubIndex		:= 16#03,
			DataLength		:= 4,
			StartReading	:= TRUE	
		);	
		Index := Index + 1;
	
	3: // Min_v is read
		IF SDO_READ.ReadDataAvailable THEN
			Label.Min_v := SHL(BYTE_TO_DWORD(SDO_READ.ReadData[3]),24) + SHL(BYTE_TO_DWORD(SDO_READ.ReadData[2]),16) + SHL(BYTE_TO_DWORD(SDO_READ.ReadData[1]),8) + BYTE_TO_DWORD(SDO_READ.ReadData[0]);				
			Index := Index + 1;
		END_IF
		
		
	4: // Start reading Max_v
		SDO_READ(	
			AdsNetID		:= GLB.ADSNetID_CAN,
			PortNr			:= 16#1000 + GLB.NodeID,
			CO_Index		:= 16#41C0,
			CO_SubIndex		:= 16#04,
			DataLength		:= 4,
			StartReading	:= TRUE	
		);	
		Index := Index + 1;
		
	5: // Max_v is read
		IF SDO_READ.ReadDataAvailable THEN
			Label.Max_v := SHL(BYTE_TO_DWORD(SDO_READ.ReadData[3]),24) + SHL(BYTE_TO_DWORD(SDO_READ.ReadData[2]),16) + SHL(BYTE_TO_DWORD(SDO_READ.ReadData[1]),8) + BYTE_TO_DWORD(SDO_READ.ReadData[0]);				
			Index := Index + 1;
		END_IF
		
		
	6: // Start reading Motor_rated_current
		SDO_READ(	
			AdsNetID		:= GLB.ADSNetID_CAN,
			PortNr			:= 16#1000 + GLB.NodeID,
			CO_Index		:= 16#41C0,
			CO_SubIndex		:= 16#05,
			DataLength		:= 4,
			StartReading	:= TRUE	
		);	
		Index := Index + 1;
		
	7: // Motor_rated_current is read
		IF SDO_READ.ReadDataAvailable THEN
			Label.Motor_rated_current := SHL(BYTE_TO_DWORD(SDO_READ.ReadData[3]),24) + SHL(BYTE_TO_DWORD(SDO_READ.ReadData[2]),16) + SHL(BYTE_TO_DWORD(SDO_READ.ReadData[1]),8) + BYTE_TO_DWORD(SDO_READ.ReadData[0]);				
			Index := Index + 1;
		END_IF
		
		
	8: // Start reading Drive_rated_current
		SDO_READ(	
			AdsNetID		:= GLB.ADSNetID_CAN,
			PortNr			:= 16#1000 + GLB.NodeID,
			CO_Index		:= 16#41C0,
			CO_SubIndex		:= 16#06,
			DataLength		:= 4,
			StartReading	:= TRUE	
		);	
		Index := Index + 1;
			
	9: // Drive_rated_current is read
		IF SDO_READ.ReadDataAvailable THEN
			Label.Drive_rated_current := SHL(BYTE_TO_DWORD(SDO_READ.ReadData[3]),24) + SHL(BYTE_TO_DWORD(SDO_READ.ReadData[2]),16) + SHL(BYTE_TO_DWORD(SDO_READ.ReadData[1]),8) + BYTE_TO_DWORD(SDO_READ.ReadData[0]);				
			Index := Index + 1;
		END_IF
		
		
	10: // Start reading Max_current
		SDO_READ(	
			AdsNetID		:= GLB.ADSNetID_CAN,
			PortNr			:= 16#1000 + GLB.NodeID,
			CO_Index		:= 16#41C0,
			CO_SubIndex		:= 16#07,
			DataLength		:= 4,
			StartReading	:= TRUE	
		);	
		Index := Index + 1;

	11: // Max_current is read
		IF SDO_READ.ReadDataAvailable THEN
			Label.Max_current := SHL(BYTE_TO_WORD(SDO_READ.ReadData[1]),8) + BYTE_TO_WORD(SDO_READ.ReadData[0]);				
			Index := Index + 1;
		END_IF
		
		
	12: // Start reading Motor_rated_torque
		SDO_READ(	
			AdsNetID		:= GLB.ADSNetID_CAN,
			PortNr			:= 16#1000 + GLB.NodeID,
			CO_Index		:= 16#41C0,
			CO_SubIndex		:= 16#08,
			DataLength		:= 4,
			StartReading	:= TRUE	
		);	
		Index := Index + 1;
	
	13: // Motor_rated_torque is read
		IF SDO_READ.ReadDataAvailable THEN
			Label.Motor_rated_torque := SHL(BYTE_TO_DWORD(SDO_READ.ReadData[3]),24) + SHL(BYTE_TO_DWORD(SDO_READ.ReadData[2]),16) + SHL(BYTE_TO_DWORD(SDO_READ.ReadData[1]),8) + BYTE_TO_DWORD(SDO_READ.ReadData[0]);				
			Index := Index + 1;
		END_IF			
		
		
	14: // Start reading Max_torque
		SDO_READ(	
			AdsNetID		:= GLB.ADSNetID_CAN,
			PortNr			:= 16#1000 + GLB.NodeID,
			CO_Index		:= 16#41C0,
			CO_SubIndex		:= 16#09,
			DataLength		:= 2,
			StartReading	:= TRUE	
		);	
		Index := Index + 1;		
		
	15: // Max_torque is read
		IF SDO_READ.ReadDataAvailable THEN
			Label.Max_torque := SHL(BYTE_TO_WORD(SDO_READ.ReadData[1]),8) + BYTE_TO_WORD(SDO_READ.ReadData[0]);
			Index := Index + 1;
		END_IF
		
		
	16: // Start reading Motor_rated_speed
		SDO_READ(	
			AdsNetID		:= GLB.ADSNetID_CAN,
			PortNr			:= 16#1000 + GLB.NodeID,
			CO_Index		:= 16#41C0,
			CO_SubIndex		:= 16#0A,
			DataLength		:= 4,
			StartReading	:= TRUE	
		);	
		Index := Index + 1;
			
	17: // Motor_rated_speed is read
		IF SDO_READ.ReadDataAvailable THEN
			Label.Motor_rated_speed := SHL(BYTE_TO_DWORD(SDO_READ.ReadData[3]),24) + SHL(BYTE_TO_DWORD(SDO_READ.ReadData[2]),16) + SHL(BYTE_TO_DWORD(SDO_READ.ReadData[1]),8) + BYTE_TO_DWORD(SDO_READ.ReadData[0]);				
			Index := Index + 1;
		END_IF
		
		
	18: // Start reading Number_of_pole_pairs
		SDO_READ(	
			AdsNetID		:= GLB.ADSNetID_CAN,
			PortNr			:= 16#1000 + GLB.NodeID,
			CO_Index		:= 16#41C0,
			CO_SubIndex		:= 16#0B,
			DataLength		:= 2,
			StartReading	:= TRUE	
		);	
		Index := Index + 1;			
		
	19: // Reading Number_of_pole_pairs, next reading Motor_torque_constant
		IF SDO_READ.ReadDataAvailable THEN
			Label.Number_of_pole_pairs := SHL(BYTE_TO_WORD(SDO_READ.ReadData[1]),8) + BYTE_TO_WORD(SDO_READ.ReadData[0]);
			Index := Index + 1;
		END_IF
		
		
	20: // Start reading Motor_torque_constant
		SDO_READ_REAL(	
				AdsNetID		:= GLB.ADSNetID_CAN,
				PortNr			:= 16#1000 + GLB.NodeID,
				CO_Index		:= 16#41C0,
				CO_SubIndex		:= 16#0C,
				StartReading	:= TRUE	
			);	
			Index := Index + 1;			
		
	21: // Motor_torque_constant is read
		IF SDO_READ_REAL.ReadDataAvailable THEN
			Label.Motor_torque_constant := SDO_READ_REAL.ReadData;
			Index := Index + 1;
		END_IF
		
		
	22: // Start reading Flux_producing_P_gain
		SDO_READ_REAL(	
			AdsNetID		:= GLB.ADSNetID_CAN,
			PortNr			:= 16#1000 + GLB.NodeID,
			CO_Index		:= 16#41C0,
			CO_SubIndex		:= 16#0D,
			StartReading	:= TRUE	
		);	
		Index := Index + 1;
					
	23: // Flux_producing_P_gain is read
		IF SDO_READ_REAL.ReadDataAvailable THEN
			Label.Flux_producing_P_gain := SDO_READ_REAL.ReadData;
			Index := Index + 1;
		END_IF
		
		
	24: // Start reading Flux_producing_I_gain
		SDO_READ_REAL(	
			AdsNetID		:= GLB.ADSNetID_CAN,
			PortNr			:= 16#1000 + GLB.NodeID,
			CO_Index		:= 16#41C0,
			CO_SubIndex		:= 16#0E,
			StartReading	:= TRUE	
		);	
		Index := Index + 1;

	25: // Flux_producing_I_gain is read
		IF SDO_READ_REAL.ReadDataAvailable THEN
			Label.Flux_producing_I_gain := SDO_READ_REAL.ReadData;
			Index := Index + 1;
		END_IF
		
		
	26: // Start reading Torque_producing_P_gain
		SDO_READ_REAL(	
			AdsNetID		:= GLB.ADSNetID_CAN,
			PortNr			:= 16#1000 + GLB.NodeID,
			CO_Index		:= 16#41C0,
			CO_SubIndex		:= 16#0F,
			StartReading	:= TRUE	
		);	
		Index := Index + 1;
		
	27: // Torque_producing_P_gain is read
		IF SDO_READ_REAL.ReadDataAvailable THEN
			Label.Torque_producing_P_gain := SDO_READ_REAL.ReadData;
			Index := Index + 1;
		END_IF
		
		
	28: // Start reading Torque_producing_I_gain
		SDO_READ_REAL(	
			AdsNetID		:= GLB.ADSNetID_CAN,
			PortNr			:= 16#1000 + GLB.NodeID,
			CO_Index		:= 16#41C0,
			CO_SubIndex		:= 16#10,
			StartReading	:= TRUE	
		);	
		Index := Index + 1;

	29: // Torque_producing_I_gain is read
		IF SDO_READ_REAL.ReadDataAvailable THEN
			Label.Torque_producing_I_gain := SDO_READ_REAL.ReadData;
			Index := Index + 1;
		END_IF
		
		
	30: // Start reading Magnetic_encoder_offset
		SDO_READ(	
			AdsNetID		:= GLB.ADSNetID_CAN,
			PortNr			:= 16#1000 + GLB.NodeID,
			CO_Index		:= 16#41C0,
			CO_SubIndex		:= 16#11,
			DataLength		:= 2,
			StartReading	:= TRUE	
		);	
		Index := Index + 1;

	31: // Magnetic_encoder_offset is read
		IF SDO_READ.ReadDataAvailable THEN
			Label.Magnetic_encoder_offset := SHL(BYTE_TO_WORD(SDO_READ.ReadData[1]),8) + BYTE_TO_WORD(SDO_READ.ReadData[0]);				
			Index := Index + 1;
		END_IF
		
		
	32: // Start reading Motor_with_brake
		SDO_READ(	
			AdsNetID		:= GLB.ADSNetID_CAN,
			PortNr			:= 16#1000 + GLB.NodeID,
			CO_Index		:= 16#41C0,
			CO_SubIndex		:= 16#12,
			DataLength		:= 2,
			StartReading	:= TRUE	
		);	
		Index := Index + 1;

	33: // Motor_with_brake is read
		IF SDO_READ.ReadDataAvailable THEN
			Label.Motor_with_brake := SHL(BYTE_TO_WORD(SDO_READ.ReadData[1]),8) + BYTE_TO_WORD(SDO_READ.ReadData[0]);				
			Index := Index + 1;
		END_IF
		
		
	34: // Start reading Encoder_mode_adjust
		SDO_READ(	
			AdsNetID		:= GLB.ADSNetID_CAN,
			PortNr			:= 16#1000 + GLB.NodeID,
			CO_Index		:= 16#41C0,
			CO_SubIndex		:= 16#13,
			DataLength		:= 2,
			StartReading	:= TRUE	
		);	
		Index := Index + 1;

	35: // Encoder_mode_adjust is read
		IF SDO_READ.ReadDataAvailable THEN
			Label.Encoder_mode_adjust := SHL(BYTE_TO_WORD(SDO_READ.ReadData[1]),8) + BYTE_TO_WORD(SDO_READ.ReadData[0]);				
			Index := Index + 1;
		END_IF
		
		
	36: // Start reading Motor_max_speed
		SDO_READ(	
			AdsNetID		:= GLB.ADSNetID_CAN,
			PortNr			:= 16#1000 + GLB.NodeID,
			CO_Index		:= 16#41C0,
			CO_SubIndex		:= 16#14,
			DataLength		:= 2,
			StartReading	:= TRUE	
		);	
		Index := Index + 1;
					
	37: // Motor_max_speed is read
		IF SDO_READ.ReadDataAvailable THEN
			Label.Motor_max_speed := SHL(BYTE_TO_WORD(SDO_READ.ReadData[1]),8) + BYTE_TO_WORD(SDO_READ.ReadData[0]);				
			Index := Index + 1;
		END_IF
				
		
	38: // Start reading Rotor_inertia
		SDO_READ_REAL(	
			AdsNetID		:= GLB.ADSNetID_CAN,
			PortNr			:= 16#1000 + GLB.NodeID,
			CO_Index		:= 16#41C0,
			CO_SubIndex		:= 16#15,
			StartReading	:= TRUE	
		);	
		Index := Index + 1;
					
	39: // Rotor_inertia is read
		IF SDO_READ_REAL.ReadDataAvailable THEN
			Label.Rotor_inertia := SDO_READ_REAL.ReadData;
			Index := Index + 1;
		END_IF
		
		
	40: // Start reading Motor_time_at_peak
		SDO_READ_REAL(	
			AdsNetID		:= GLB.ADSNetID_CAN,
			PortNr			:= 16#1000 + GLB.NodeID,
			CO_Index		:= 16#41C0,
			CO_SubIndex		:= 16#17,
			StartReading	:= TRUE	
		);	
		Index := Index + 1;
					
	41: // Motor_time_at_peak is read
		IF SDO_READ_REAL.ReadDataAvailable THEN
			Label.Motor_time_at_peak := SDO_READ_REAL.ReadData;
			Index := Index + 1;
		END_IF
		
		
	42: // Start reading Drive_time_at_peak
		SDO_READ_REAL(	
			AdsNetID		:= GLB.ADSNetID_CAN,
			PortNr			:= 16#1000 + GLB.NodeID,
			CO_Index		:= 16#41C0,
			CO_SubIndex		:= 16#18,
			StartReading	:= TRUE	
		);	
		Index := Index + 1;
		
	43: // Drive_time_at_peak is read
		IF SDO_READ_REAL.ReadDataAvailable THEN
			Label.Drive_time_at_peak := SDO_READ_REAL.ReadData;
			Index := Index + 1;
		END_IF
		
		
	44: // Start reading Singleturn_resolution
		SDO_READ(	
			AdsNetID		:= GLB.ADSNetID_CAN,
			PortNr			:= 16#1000 + GLB.NodeID,
			CO_Index		:= 16#41C0,
			CO_SubIndex		:= 16#19,
			DataLength		:= 1,
			StartReading	:= TRUE	
		);	
		Index := Index + 1;
					
	45: // Singleturn_resolution is read 
		IF SDO_READ.ReadDataAvailable THEN
			Label.Singleturn_resolution := SDO_READ.ReadData[0];				
			Index := Index + 1;
		END_IF		
		
		
	46: // Start reading Multiturn_resolution
		SDO_READ(	
			AdsNetID		:= GLB.ADSNetID_CAN,
			PortNr			:= 16#1000 + GLB.NodeID,
			CO_Index		:= 16#41C0,
			CO_SubIndex		:= 16#1A,
			DataLength		:= 1,
			StartReading	:= TRUE	
		);	
		Index := Index + 1;
			
	47: // Multiturn_resolution is read
		IF SDO_READ.ReadDataAvailable THEN
			Label.Multiturn_resolution := SDO_READ.ReadData[0];	
			Index := 255;
		END_IF		
				
		
	255: // Finished 
		Label_Out := Label;
		Finished := TRUE;
				
		
	ELSE
		Index := 255;
			
END_CASE

END_FUNCTION_BLOCK

// ---- POUs/FB/Basic/FB_SDO_READ_REAL.TcPOU
FUNCTION_BLOCK FB_SDO_READ_REAL
VAR_INPUT
	ADSNetID		: STRING(23); 	(* The AMSNetID addresses the EL6751. Can be empty if only one local single channel card is present*)
	PortNr			: WORD;	 		(* This Port No. addresses the CANopen Node (see System Manager) *)
	CO_Index		: DWORD; 		(* This is the Index of the CANopen Object Dictionary Entry*)
	CO_SubIndex		: DWORD; 		(* This is the Sub-Index of the CANopen Object Dictionary Entry*)
	StartReading	: BOOL;  		(* only reset to FALSE after ReadDataAvailable=TRUE*)
END_VAR
VAR_OUTPUT
	ReadData		: REAL;
	ReadDataAvailable	: BOOL;
	Error			: DWORD;
END_VAR
VAR
	state			: BYTE 	:= 0;
	ADSREAD			: ADSREAD;
END_VAR

CASE
state OF
0:
	IF StartReading THEN
		ReadDataAvailable := FALSE;
		Error := 0;
		ADSRead(
			NETID		:= ADSNetID,
			PORT		:= PortNr,
			IDXGRP		:= CO_Index,
			IDXOFFS		:= CO_SubIndex,
			LEN			:= 4,
			DESTADDR	:= ADR(ReadData),
			READ		:= TRUE,
			TMOUT		:= T#100MS
		);

		IF ADSRead.err THEN
			state := 2;
			ReadDataAvailable := TRUE;
			Error := ADSRead.ErrId;
		ELSE
			state := 1;
		END_IF
	ELSE
		ADSRead(
			NETID		:= ADSNetID,
			PORT		:= PortNr,
			IDXGRP		:= CO_Index,
			IDXOFFS		:= CO_SubIndex,
			LEN			:= 4,
			DESTADDR	:= ADR(ReadData),
			READ		:= FALSE,
			TMOUT 		:= T#100MS
		);
	END_IF
	
1:
	ADSRead(READ:= FALSE);
	IF ADSRead.err THEN
		state := 2;
		ReadDataAvailable := TRUE;
		Error := ADSRead.ErrId;
	ELSE
		IF NOT ADSRead.busy THEN
			state := 2;
			ReadDataAvailable := TRUE;
		END_IF
	END_IF
	
2:
	ADSRead(READ:= FALSE);
	state := 0;
	
END_CASE

END_FUNCTION_BLOCK

// ---- POUs/Encoder_Alignment.TcPOU
FUNCTION_BLOCK Encoder_Alignment
VAR_INPUT
	Start 			: BOOL;
	Current_State 	: E_Statemachine_State;	
	Statusword		: WORD;	
END_VAR
VAR_OUTPUT
	Controlword 	: WORD;
	Encoder_offset	: WORD;
	Finished		: BOOL;
END_VAR
VAR
	Index 			: BYTE := 0;
	
	SDO_WRITE		: FB_SDO_WRITE;
	WriteData		: ARRAY [0..255] OF BYTE;
	
	SDO_READ		: FB_SDO_READ;
	ReadStart		: BOOL;
	ReadError		: DWORD;
	ReadData		: ARRAY [0..255] OF BYTE;
	
	fbTonDelay		: TON;
	Start_old		: BOOL := FALSE;
END_VAR

// Restart after complete run
IF NOT Start_old AND Start THEN
	Index := 0;
	Finished := FALSE;
END_IF


CASE Index OF	
	0: // Switch to state 'Switch on disabled'
		IF (Start) THEN
			Controlword := CONTROLWORD_STATE_CHANGE(Current_State, E_Statemachine_State.Switch_on_disabled);
			IF (Current_State = E_Statemachine_State.Switch_on_disabled) THEN			
				Index := Index + 2;
			ELSE
				Index := Index + 1;		
			END_IF
		END_IF
		
			
	1: // Wait for 'Switch on disabled'
		Controlword := CONTROLWORD_STATE_CHANGE(Current_State, E_Statemachine_State.Switch_on_disabled);	
		IF (Current_State = E_Statemachine_State.Switch_on_disabled) THEN			
			Index := Index + 1;		
		END_IF
					
		
	2: // Set Mode of operation
		PDO.Mode_of_operation := E_Mode_of_operation.Phasing_mode;	
		Controlword := CONTROLWORD_STATE_CHANGE(Current_State, E_Statemachine_State.Switch_on_disabled);				
		IF (PDO.Mode_of_operation_display = E_Mode_of_operation.Phasing_mode) THEN			
			Index := Index + 1;		
		END_IF

		
	3: // Start
		Controlword := CONTROLWORD_STATE_CHANGE(Current_State, E_Statemachine_State.Operation_enabled);	
		IF ((Current_State = E_Statemachine_State.Operation_enabled) AND ((Statusword AND E_Statusword_Bits.Manufacturer_specific_3) <> 0)) THEN			
			Index := Index + 1;		
		END_IF
		
		
	4: // Wait for finish
		Controlword := CONTROLWORD_STATE_CHANGE(Current_State, E_Statemachine_State.Operation_enabled);			
		IF ((Statusword AND E_Statusword_Bits.Manufacturer_specific_3) = 0) THEN			
			Index := Index + 1;		
		END_IF
	
		
	5: // Switch State to 'Switch on disabled'
		Controlword := CONTROLWORD_STATE_CHANGE(Current_State, E_Statemachine_State.Switch_on_disabled);	
		IF (Current_State = E_Statemachine_State.Switch_on_disabled) THEN			
			Index := Index + 1;
		END_IF
		
		
	6: // Save		
		Controlword := CONTROLWORD_STATE_CHANGE(Current_State, E_Statemachine_State.Switch_on_disabled);	
		WriteData[0] := 16#73;	// s
		WriteData[1] := 16#61;	// a
		WriteData[2] := 16#76;	// v
		WriteData[3] := 16#65;	// e		
		SDO_WRITE(	
			AdsNetID		:= GLB.ADSNetID_CAN,
			PortNr			:= 16#1000 + GLB.NodeID,
			CO_Index		:= 16#1010,
			CO_SubIndex		:= 16#04,
			DataLength		:= 4,
			WriteData		:= WriteData,
			StartWriting	:= TRUE	
		);	
		Index := Index + 1;		

		
	7: // Wait for finish sdo transfer	
		Controlword := CONTROLWORD_STATE_CHANGE(Current_State, E_Statemachine_State.Switch_on_disabled);	
		SDO_WRITE(StartWriting := FALSE);
		IF SDO_WRITE.WriteDataFinished THEN
			Index := Index + 1;			
		END_IF		
		
		
	8: // Wait 500 ms for save process
		Controlword := CONTROLWORD_STATE_CHANGE(Current_State, E_Statemachine_State.Switch_on_disabled);	
		fbTonDelay(IN := TRUE, PT:= T#500MS);
		IF fbTonDelay.Q THEN
			fbTonDelay(IN := FALSE);
			Index := Index + 1;	
		END_IF
		
		
	9: // Read the alignment offset
		Controlword := CONTROLWORD_STATE_CHANGE(Current_State, E_Statemachine_State.Switch_on_disabled);	
		SDO_READ(	
			AdsNetID		:= GLB.ADSNetID_CAN,
			PortNr			:= 16#1000 + GLB.NodeID,
			CO_Index		:= 16#41C0,
			CO_SubIndex		:= 16#11,
			DataLength		:= 2,
			StartReading	:= TRUE	
		);	
		Index := Index + 1;	
		
		
	10: // Wait for finish sdo transfer
		Controlword := CONTROLWORD_STATE_CHANGE(Current_State, E_Statemachine_State.Switch_on_disabled);	
		SDO_Read(StartReading := FALSE);
		IF SDO_WRITE.WriteDataFinished THEN			
			Encoder_offset := SHL(BYTE_TO_WORD(SDO_READ.ReadData[1]),8) + BYTE_TO_WORD(SDO_READ.ReadData[0]);
			Index := 255;			
		END_IF	
			
		
	255: // Finished 
		Controlword := CONTROLWORD_STATE_CHANGE(Current_State, E_Statemachine_State.Switch_on_disabled);	
		FINISHED := TRUE;
				
		
	ELSE
		Index := 255;
			
END_CASE


Start_old := Start;

END_FUNCTION_BLOCK

// ---- POUs/CONTROLWORD_STATE_CHANGE.TcPOU
FUNCTION CONTROLWORD_STATE_CHANGE : WORD
VAR_INPUT
	Current_State 		: E_Statemachine_State;
	Target_State 		: E_Statemachine_State;	
END_VAR
VAR
	Controlword 		: WORD;
END_VAR

CASE Current_State OF
    E_Statemachine_State.Not_ready_to_switch_on:		// Wait for 'Switch on disabled'
		Controlword := E_Statemachine_Transition_Controlword.Switch_on_disabled;

	E_Statemachine_State.Switch_on_disabled:
		CASE Target_State OF
			E_Statemachine_State.Ready_to_switch_on:	Controlword := E_Statemachine_Transition_Controlword.Ready_to_switch_on;				
			E_Statemachine_State.Switched_on:			Controlword := E_Statemachine_Transition_Controlword.Ready_to_switch_on;				
			E_Statemachine_State.Operation_enabled:		Controlword := E_Statemachine_Transition_Controlword.Ready_to_switch_on;				
		ELSE
			Controlword := E_Statemachine_Transition_Controlword.Switch_on_disabled;			
		END_CASE

	E_Statemachine_State.Ready_to_switch_on:
		CASE Target_State OF
			E_Statemachine_State.Switch_on_disabled:	Controlword := E_Statemachine_Transition_Controlword.Switch_on_disabled;			
			E_Statemachine_State.Switched_on:			Controlword := E_Statemachine_Transition_Controlword.Switched_on;			
			E_Statemachine_State.Operation_enabled:		Controlword := E_Statemachine_Transition_Controlword.Switched_on;					
		ELSE
			Controlword := E_Statemachine_Transition_Controlword.Ready_to_switch_on;			
		END_CASE
				
	E_Statemachine_State.Switched_on:
		CASE Target_State OF
			E_Statemachine_State.Switch_on_disabled:	Controlword := E_Statemachine_Transition_Controlword.Switch_on_disabled;		
			E_Statemachine_State.Ready_to_switch_on:	Controlword := E_Statemachine_Transition_Controlword.Ready_to_switch_on;	
			E_Statemachine_State.Operation_enabled:		Controlword := E_Statemachine_Transition_Controlword.Operation_enabled;				
		ELSE
			CONTROLWORD_STATE_CHANGE := E_Statemachine_Transition_Controlword.Switched_on;				
		END_CASE
		
	E_Statemachine_State.Operation_enabled:
		CASE Target_State OF
			E_Statemachine_State.Switch_on_disabled:	Controlword := E_Statemachine_Transition_Controlword.Switch_on_disabled;		
			E_Statemachine_State.Ready_to_switch_on:	Controlword := E_Statemachine_Transition_Controlword.Ready_to_switch_on;	
			E_Statemachine_State.Switched_on:			Controlword := E_Statemachine_Transition_Controlword.Switched_on;		
			E_Statemachine_State.Quick_stop_active:		Controlword := E_Statemachine_Transition_Controlword.Quick_stop_active;				
		ELSE
			Controlword := E_Statemachine_Transition_Controlword.Operation_enabled;	;			
		END_CASE
		
	E_Statemachine_State.Quick_stop_active:				
		CASE Target_State OF
			E_Statemachine_State.Switch_on_disabled:	Controlword := E_Statemachine_Transition_Controlword.Switch_on_disabled;		
			E_Statemachine_State.Ready_to_switch_on:	Controlword := E_Statemachine_Transition_Controlword.Switch_on_disabled;	
			E_Statemachine_State.Switched_on:			Controlword := E_Statemachine_Transition_Controlword.Switch_on_disabled;	
			E_Statemachine_State.Operation_enabled:		Controlword := E_Statemachine_Transition_Controlword.Switch_on_disabled;	// Not recommennded to support to switch back directly			
		ELSE
			Controlword := 16#2;			
		END_CASE
		
	E_Statemachine_State.Fault_reaction_active:			// Wait for 'Fault'
		Controlword := E_Statemachine_Transition_Controlword.Switch_on_disabled;
		
	E_Statemachine_State.Fault:
		CASE Target_State OF
 			E_Statemachine_State.Switch_on_disabled, E_Statemachine_State.Ready_to_switch_on, E_Statemachine_State.Switched_on, E_Statemachine_State.Operation_enabled:
				// Toggle the Fault reset bit
				IF PDO.Controlword = E_Statemachine_Transition_Controlword.Faultreset_step_2 THEN	Controlword := E_Statemachine_Transition_Controlword.Faultreset_step_1; ELSE Controlword := E_Statemachine_Transition_Controlword.Faultreset_step_2; END_IF
		ELSE
			Controlword := E_Statemachine_Transition_Controlword.Switch_on_disabled;
		END_CASE;
	
ELSE
    Controlword := 16#0;
	
END_CASE;

// Return the new controlword
CONTROLWORD_STATE_CHANGE := Controlword;

END_FUNCTION

// ---- POUs/Homing_Mode.TcPOU
FUNCTION_BLOCK Homing_Mode
VAR_INPUT
	NodeID				: BYTE; (* This Port No. addresses the CANopen Node (see System Manager) *)
	Start 				: BOOL;
	Current_State 		: E_Statemachine_State;	
	Statusword			: WORD;	
	Homing_parameters	: ST_Homing_parameters;
END_VAR
VAR_OUTPUT
	Controlword 		: WORD;
	Mode_of_operation 	: E_Mode_of_operation	:= E_Mode_of_operation.No_mode_active;
	Finished			: BOOL;
END_VAR
VAR
	Index 			: BYTE := 0;
	
	SDO_WRITE		: FB_SDO_WRITE;
	WriteData		: ARRAY [0..255] OF BYTE;
	
	SDO_READ		: FB_SDO_READ;
	ReadStart		: BOOL;
	ReadError		: DWORD;
	ReadData		: ARRAY [0..255] OF BYTE;
	
	fbTonDelay		: TON;
	Start_old		: BOOL := FALSE;
END_VAR

